QRS_NEXT_CUT()
PTP {E1 35457.209,E2 35457.209}
PTP {X 0,Y 759.903,A -85,B 0,C 180,E1 35457.209,E2 35457.209,E3 0,E4 0,E5 0,E6 0}
QRS_SPEED_INIT()
LIN {X 0,Y 759.903,Z 1305,A -85,B 0,C 180,E1 35457.209,E2 35457.209,E3 0,E4 0,E5 0,E6 0} C_VEL
LIN {X 0,Y 759.903,Z 603.404,A -85,B 0,C 180,E1 35457.209,E2 35457.209} C_VEL
LIN {X 0,Y 759.903,Z 595.326,A -85,B 0,C 180,E1 35457.209,E2 35457.209} C_VEL
LIN {X 0,Y 759.893,Z 593.326,A -85,B 0,C 180,E1 35457.058,E2 35457.058} C_VEL
LIN {X 0,Y 759.912,Z 593.326,A -85,B 0,C 180,E1 35454.261,E2 35454.261} C_VEL
LIN {X 0,Y 759.899,Z 593.323,A -85,B 0,C 180,E1 35451.373,E2 35451.373} C_VEL
LIN {X 0,Y 759.889,Z 593.322,A -85,B 0,C 180,E1 35448.539,E2 35448.539} C_VEL
LIN {X 0,Y 759.901,Z 593.322,A -85,B 0,C 180,E1 35445.756,E2 35445.756} C_VEL
LIN {X 0,Y 759.919,Z 593.324,A -85,B 0,C 180,E1 35442.858,E2 35442.858} C_VEL
LIN {X 0,Y 759.909,Z 593.326,A -85,B 0,C 180,E1 35439.96,E2 35439.96} C_VEL
LIN {X 0,Y 759.889,Z 593.323,A -85,B 0,C 180,E1 35437.159,E2 35437.159} C_VEL
LIN {X 0,Y 759.903,Z 593.32,A -85,B 0,C 180,E1 35434.33,E2 35434.33} C_VEL
LIN {X 0,Y 759.916,Z 593.32,A -85,B 0,C 180,E1 35431.354,E2 35431.354} C_VEL
LIN {X 0,Y 759.914,Z 593.321,A -85,B 0,C 180,E1 35428.331,E2 35428.331} C_VEL
LIN {X 0,Y 759.905,Z 593.327,A -85,B 0,C 180,E1 35425.451,E2 35425.451} C_VEL
LIN {X 0,Y 759.89,Z 593.326,A -85,B 0,C 180,E1 35422.656,E2 35422.656} C_VEL
LIN {X 0,Y 759.912,Z 593.32,A -85,B 0,C 180,E1 35419.853,E2 35419.853} C_VEL
LIN {X 0,Y 759.91,Z 593.319,A -85,B 0,C 180,E1 35416.826,E2 35416.826} C_VEL
LIN {X 0,Y 759.911,Z 593.32,A -85,B 0,C 180,E1 35413.795,E2 35413.795} C_VEL
LIN {X 0,Y 759.892,Z 593.325,A -85,B 0,C 180,E1 35410.939,E2 35410.939} C_VEL
LIN {X 0,Y 759.898,Z 593.327,A -85,B 0,C 180,E1 35408.2,E2 35408.2} C_VEL
LIN {X 0,Y 759.916,Z 593.321,A -85,B 0,C 180,E1 35405.282,E2 35405.282} C_VEL
LIN {X 0,Y 759.911,Z 593.32,A -85,B 0,C 180,E1 35402.289,E2 35402.289} C_VEL
LIN {X 0,Y 759.904,Z 593.321,A -85,B 0,C 180,E1 35399.305,E2 35399.305} C_VEL
LIN {X 0,Y 759.909,Z 593.575,A -85,B 0,C 180,E1 35398.059,E2 35398.059} C_VEL
LIN {X 0,Y 759.899,Z 638.776,A -85,B 0,C 180,E1 35395.191,E2 35395.191} C_VEL
LIN {X 0,Y 759.89,Z 682.695,A -85,B 0,C 180,E1 35392.472,E2 35392.472} C_VEL
LIN {X 0,Y 759.915,Z 727.991,A -85,B 0,C 180,E1 35389.723,E2 35389.723} C_VEL
LIN {X 0,Y 759.912,Z 778.002,A -85,B 0,C 180,E1 35386.746,E2 35386.746} C_VEL
LIN {X 0,Y 759.9,Z 826.73,A -85,B 0,C 180,E1 35383.893,E2 35383.893} C_VEL
LIN {X 0,Y 759.916,Z 830.801,A -85,B 0,C 180,E1 35383.665,E2 35383.665} C_VEL
LIN {X 0,Y 759.906,Z 999.951,A -85,B 0,C 180,E1 35382.036,E2 35382.036} C_VEL
LIN {X 0,Y 759.914,Z 1017.524,A -85,B 0,C 180,E1 35381.728,E2 35381.728} C_VEL
LIN {X 0,Y 759.905,Z 1033.905,A -85,B 0,C 180,E1 35381.305,E2 35381.305} C_VEL
LIN {X 0,Y 759.911,Z 1050.473,A -85,B 0,C 180,E1 35380.729,E2 35380.729} C_VEL
LIN {X 0,Y 759.918,Z 1065.925,A -85,B 0,C 180,E1 35380.039,E2 35380.039} C_VEL
LIN {X 0,Y 759.918,Z 1080.253,A -85,B 0,C 180,E1 35379.236,E2 35379.236} C_VEL
LIN {X 0,Y 759.918,Z 1093.584,A -85,B 0,C 180,E1 35378.319,E2 35378.319} C_VEL
LIN {X 0,Y 759.918,Z 1105.366,A -85,B 0,C 180,E1 35377.332,E2 35377.332} C_VEL
LIN {X 0,Y 759.919,Z 1115.725,A -85,B 0,C 180,E1 35376.269,E2 35376.269} C_VEL
LIN {X 0,Y 759.915,Z 1124.926,A -85,B 0,C 180,E1 35375.088,E2 35375.088} C_VEL
LIN {X 0,Y 759.916,Z 1132.481,A -85,B 0,C 180,E1 35373.847,E2 35373.847} C_VEL
LIN {X 0,Y 759.914,Z 1138.296,A -85,B 0,C 180,E1 35372.563,E2 35372.563} C_VEL
LIN {X 0,Y 759.913,Z 1142.253,A -85,B 0,C 180,E1 35371.281,E2 35371.281} C_VEL
LIN {X 0,Y 759.916,Z 1144.493,A -85,B 0,C 180,E1 35369.924,E2 35369.924} C_VEL
LIN {X 0,Y 759.915,Z 1144.892,A -85,B 0,C 180,E1 35368.566,E2 35368.566} C_VEL
LIN {X 0,Y 759.912,Z 1143.454,A -85,B 0,C 180,E1 35367.208,E2 35367.208} C_VEL
LIN {X 0,Y 759.918,Z 1140.29,A -85,B 0,C 180,E1 35365.925,E2 35365.925} C_VEL
LIN {X 0,Y 759.914,Z 1135.319,A -85,B 0,C 180,E1 35364.639,E2 35364.639} C_VEL
LIN {X 0,Y 759.914,Z 1128.391,A -85,B 0,C 180,E1 35363.35,E2 35363.35} C_VEL
LIN {X 0,Y 759.916,Z 1119.844,A -85,B 0,C 180,E1 35362.134,E2 35362.134} C_VEL
LIN {X 0,Y 759.917,Z 1109.619,A -85,B 0,C 180,E1 35360.991,E2 35360.991} C_VEL
LIN {X 0,Y 759.917,Z 1097.777,A -85,B 0,C 180,E1 35359.92,E2 35359.92} C_VEL
LIN {X 0,Y 759.917,Z 1085.153,A -85,B 0,C 180,E1 35358.987,E2 35358.987} C_VEL
LIN {X 0,Y 759.918,Z 1071.315,A -85,B 0,C 180,E1 35358.154,E2 35358.154} C_VEL
LIN {X 0,Y 759.913,Z 1056.24,A -85,B 0,C 180,E1 35357.421,E2 35357.421} C_VEL
LIN {X 0,Y 759.91,Z 1039.961,A -85,B 0,C 180,E1 35356.797,E2 35356.797} C_VEL
LIN {X 0,Y 759.908,Z 1023.505,A -85,B 0,C 180,E1 35356.318,E2 35356.318} C_VEL
LIN {X 0,Y 759.909,Z 1006.36,A -85,B 0,C 180,E1 35355.969,E2 35355.969} C_VEL
LIN {X 0,Y 759.906,Z 987.058,A -85,B 0,C 180,E1 35355.735,E2 35355.735} C_VEL
LIN {X 0,Y 759.911,Z 830.448,A -85,B 0,C 180,E1 35354.233,E2 35354.233} C_VEL
LIN {X 0,Y 759.914,Z 779.85,A -85,B 0,C 180,E1 35351.273,E2 35351.273} C_VEL
LIN {X 0,Y 759.905,Z 729.874,A -85,B 0,C 180,E1 35348.299,E2 35348.299} C_VEL
LIN {X 0,Y 759.889,Z 684.484,A -85,B 0,C 180,E1 35345.548,E2 35345.548} C_VEL
LIN {X 0,Y 759.904,Z 640.226,A -85,B 0,C 180,E1 35342.81,E2 35342.81} C_VEL
LIN {X 0,Y 759.907,Z 594.516,A -85,B 0,C 180,E1 35339.912,E2 35339.912} C_VEL
LIN {X 0,Y 759.91,Z 593.318,A -85,B 0,C 180,E1 35339.824,E2 35339.824} C_VEL
LIN {X 0,Y 759.915,Z 593.322,A -85,B 0,C 180,E1 35336.809,E2 35336.809} C_VEL
LIN {X 0,Y 759.891,Z 593.317,A -85,B 0,C 180,E1 35333.972,E2 35333.972} C_VEL
LIN {X 0,Y 759.918,Z 593.327,A -85,B 0,C 180,E1 35331.124,E2 35331.124} C_VEL
LIN {X 0,Y 759.906,Z 593.315,A -85,B 0,C 180,E1 35328.251,E2 35328.251} C_VEL
LIN {X 0,Y 759.913,Z 593.328,A -85,B 0,C 180,E1 35325.255,E2 35325.255} C_VEL
LIN {X 0,Y 759.906,Z 593.315,A -85,B 0,C 180,E1 35322.251,E2 35322.251} C_VEL
LIN {X 0,Y 759.91,Z 593.328,A -85,B 0,C 180,E1 35319.313,E2 35319.313} C_VEL
LIN {X 0,Y 759.889,Z 593.318,A -85,B 0,C 180,E1 35316.488,E2 35316.488} C_VEL
LIN {X 0,Y 759.914,Z 593.324,A -85,B 0,C 180,E1 35313.602,E2 35313.602} C_VEL
LIN {X 0,Y 759.911,Z 593.315,A -85,B 0,C 180,E1 35310.612,E2 35310.612} C_VEL
LIN {X 0,Y 759.918,Z 593.327,A -85,B 0,C 180,E1 35307.591,E2 35307.591} C_VEL
LIN {X 0,Y 759.91,Z 593.353,A -85,B 0,C 180,E1 35306.575,E2 35306.575} C_VEL
LIN {X 0,Y 759.889,Z 601.331,A -85,B 0,C 180,E1 35305.967,E2 35305.967} C_VEL
LIN {X 0,Y 759.915,Z 858.573,A -85,B 0,C 180,E1 35303.276,E2 35303.276} C_VEL
LIN {X 0,Y 759.913,Z 946.529,A -85,B 0,C 180,E1 35302.35,E2 35302.35} C_VEL
LIN {X 0,Y 759.909,Z 970.175,A -85,B 0,C 180,E1 35301.964,E2 35301.964} C_VEL
LIN {X 0,Y 759.908,Z 991.488,A -85,B 0,C 180,E1 35301.489,E2 35301.489} C_VEL
LIN {X 0,Y 759.898,Z 1013.758,A -85,B 0,C 180,E1 35300.851,E2 35300.851} C_VEL
LIN {X 0,Y 759.918,Z 1033.44,A -85,B 0,C 180,E1 35300.166,E2 35300.166} C_VEL
LIN {X 0,Y 759.919,Z 1054.673,A -85,B 0,C 180,E1 35299.285,E2 35299.285} C_VEL
LIN {X 0,Y 759.914,Z 1074.389,A -85,B 0,C 180,E1 35298.329,E2 35298.329} C_VEL
LIN {X 0,Y 759.917,Z 1093.916,A -85,B 0,C 180,E1 35297.221,E2 35297.221} C_VEL
LIN {X 0,Y 759.911,Z 1112.133,A -85,B 0,C 180,E1 35296.041,E2 35296.041} C_VEL
LIN {X 0,Y 759.913,Z 1129.871,A -85,B 0,C 180,E1 35294.711,E2 35294.711} C_VEL
LIN {X 0,Y 759.909,Z 1146.093,A -85,B 0,C 180,E1 35293.313,E2 35293.313} C_VEL
LIN {X 0,Y 759.909,Z 1161,A -85,B 0,C 180,E1 35291.845,E2 35291.845} C_VEL
LIN {X 0,Y 759.899,Z 1173.75,A -85,B 0,C 180,E1 35290.385,E2 35290.385} C_VEL
LIN {X 0,Y 759.909,Z 1186.404,A -85,B 0,C 180,E1 35288.703,E2 35288.703} C_VEL
LIN {X 0,Y 759.911,Z 1196.1,A -85,B 0,C 180,E1 35287.181,E2 35287.181} C_VEL
LIN {X 0,Y 759.896,Z 1205.307,A -85,B 0,C 180,E1 35285.436,E2 35285.436} C_VEL
LIN {X 0,Y 759.903,Z 1211.799,A -85,B 0,C 180,E1 35283.923,E2 35283.923} C_VEL
LIN {X 0,Y 759.915,Z 1217.779,A -85,B 0,C 180,E1 35282.111,E2 35282.111} C_VEL
LIN {X 0,Y 759.917,Z 1221.69,A -85,B 0,C 180,E1 35280.452,E2 35280.452} C_VEL
LIN {X 0,Y 759.91,Z 1224.098,A -85,B 0,C 180,E1 35278.718,E2 35278.718} C_VEL
LIN {X 0,Y 759.909,Z 1224.976,A -85,B 0,C 180,E1 35277.058,E2 35277.058} C_VEL
LIN {X 0,Y 759.91,Z 1224.211,A -85,B 0,C 180,E1 35275.321,E2 35275.321} C_VEL
LIN {X 0,Y 759.894,Z 1221.944,A -85,B 0,C 180,E1 35273.578,E2 35273.578} C_VEL
LIN {X 0,Y 759.917,Z 1218.072,A -85,B 0,C 180,E1 35271.906,E2 35271.906} C_VEL
LIN {X 0,Y 759.914,Z 1212.453,A -85,B 0,C 180,E1 35270.151,E2 35270.151} C_VEL
LIN {X 0,Y 759.906,Z 1205.614,A -85,B 0,C 180,E1 35268.54,E2 35268.54} C_VEL
LIN {X 0,Y 759.914,Z 1196.782,A -85,B 0,C 180,E1 35266.842,E2 35266.842} C_VEL
LIN {X 0,Y 759.897,Z 1186.955,A -85,B 0,C 180,E1 35265.288,E2 35265.288} C_VEL
LIN {X 0,Y 759.907,Z 1174.745,A -85,B 0,C 180,E1 35263.645,E2 35263.645} C_VEL
LIN {X 0,Y 759.914,Z 1162.457,A -85,B 0,C 180,E1 35262.226,E2 35262.226} C_VEL
LIN {X 0,Y 759.916,Z 1147.367,A -85,B 0,C 180,E1 35260.715,E2 35260.715} C_VEL
LIN {X 0,Y 759.915,Z 1131.348,A -85,B 0,C 180,E1 35259.314,E2 35259.314} C_VEL
LIN {X 0,Y 759.917,Z 1113.604,A -85,B 0,C 180,E1 35257.976,E2 35257.976} C_VEL
LIN {X 0,Y 759.917,Z 1094.916,A -85,B 0,C 180,E1 35256.75,E2 35256.75} C_VEL
LIN {X 0,Y 759.919,Z 1076.273,A -85,B 0,C 180,E1 35255.679,E2 35255.679} C_VEL
LIN {X 0,Y 759.916,Z 1055.929,A -85,B 0,C 180,E1 35254.682,E2 35254.682} C_VEL
LIN {X 0,Y 759.918,Z 1034.648,A -85,B 0,C 180,E1 35253.788,E2 35253.788} C_VEL
LIN {X 0,Y 759.902,Z 1014.583,A -85,B 0,C 180,E1 35253.087,E2 35253.087} C_VEL
LIN {X 0,Y 759.918,Z 993.181,A -85,B 0,C 180,E1 35252.462,E2 35252.462} C_VEL
LIN {X 0,Y 759.906,Z 971.975,A -85,B 0,C 180,E1 35251.982,E2 35251.982} C_VEL
LIN {X 0,Y 759.915,Z 949.573,A -85,B 0,C 180,E1 35251.598,E2 35251.598} C_VEL
LIN {X 0,Y 759.914,Z 903.373,A -85,B 0,C 180,E1 35251.095,E2 35251.095} C_VEL
LIN {X 0,Y 759.913,Z 631.659,A -85,B 0,C 180,E1 35248.265,E2 35248.265} C_VEL
LIN {X 0,Y 759.893,Z 600.869,A -85,B 0,C 180,E1 35247.93,E2 35247.93} C_VEL
LIN {X 0,Y 759.911,Z 593.322,A -85,B 0,C 180,E1 35247.307,E2 35247.307} C_VEL
LIN {X 0,Y 759.897,Z 593.322,A -85,B 0,C 180,E1 35244.344,E2 35244.344} C_VEL
LIN {X 0,Y 759.891,Z 593.324,A -85,B 0,C 180,E1 35241.529,E2 35241.529} C_VEL
LIN {X 0,Y 759.902,Z 593.328,A -85,B 0,C 180,E1 35238.706,E2 35238.706} C_VEL
LIN {X 0,Y 759.913,Z 593.325,A -85,B 0,C 180,E1 35236.888,E2 35236.888} C_VEL
LIN {X 0,Y 759.918,Z 654.539,A -85,B 0,C 180,E1 35234.851,E2 35234.851} C_VEL
LIN {X 0,Y 759.92,Z 699.236,A -85,B 0,C 180,E1 35233.202,E2 35233.202} C_VEL
LIN {X 0,Y 759.92,Z 738.808,A -85,B 0,C 180,E1 35231.589,E2 35231.589} C_VEL
LIN {X 0,Y 759.917,Z 752.824,A -85,B 0,C 180,E1 35230.89,E2 35230.89} C_VEL
LIN {X 0,Y 759.908,Z 764.753,A -85,B 0,C 180,E1 35230.139,E2 35230.139} C_VEL
LIN {X 0,Y 759.908,Z 773.509,A -85,B 0,C 180,E1 35229.432,E2 35229.432} C_VEL
LIN {X 0,Y 759.893,Z 779.468,A -85,B 0,C 180,E1 35228.781,E2 35228.781} C_VEL
LIN {X 0,Y 759.895,Z 782.672,A -85,B 0,C 180,E1 35228.203,E2 35228.203} C_VEL
LIN {X 0,Y 759.891,Z 783.283,A -85,B 0,C 180,E1 35227.82,E2 35227.82} C_VEL
LIN {X 0,Y 759.909,Z 782.173,A -85,B 0,C 180,E1 35227.493,E2 35227.493} C_VEL
LIN {X 0,Y 759.899,Z 779.495,A -85,B 0,C 180,E1 35227.243,E2 35227.243} C_VEL
LIN {X 0,Y 759.891,Z 775.795,A -85,B 0,C 180,E1 35227.089,E2 35227.089} C_VEL
LIN {X 0,Y 759.889,Z 769.468,A -85,B 0,C 180,E1 35226.992,E2 35226.992} C_VEL
LIN {X 0,Y 759.889,Z 593.325,A -85,B 0,C 180,E1 35226.966,E2 35226.966} C_VEL
LIN {X 0,Y 759.9,Z 593.351,A -85,B 0,C 180,E1 35224.136,E2 35224.136} C_VEL
LIN {X 0,Y 759.915,Z 633.667,A -85,B 0,C 180,E1 35221.404,E2 35221.404} C_VEL
LIN {X 0,Y 759.908,Z 669.855,A -85,B 0,C 180,E1 35219.026,E2 35219.026} C_VEL
LIN {X 0,Y 759.91,Z 945.711,A -85,B 0,C 180,E1 35216.145,E2 35216.145} C_VEL
LIN {X 0,Y 759.903,Z 1017.761,A -85,B 0,C 180,E1 35215.381,E2 35215.381} C_VEL
LIN {X 0,Y 759.916,Z 1040.309,A -85,B 0,C 180,E1 35215.006,E2 35215.006} C_VEL
LIN {X 0,Y 759.901,Z 1060.837,A -85,B 0,C 180,E1 35214.55,E2 35214.55} C_VEL
LIN {X 0,Y 759.918,Z 1083.358,A -85,B 0,C 180,E1 35213.908,E2 35213.908} C_VEL
LIN {X 0,Y 759.919,Z 1103.501,A -85,B 0,C 180,E1 35213.209,E2 35213.209} C_VEL
LIN {X 0,Y 759.917,Z 1124.653,A -85,B 0,C 180,E1 35212.331,E2 35212.331} C_VEL
LIN {X 0,Y 759.913,Z 1144.352,A -85,B 0,C 180,E1 35211.376,E2 35211.376} C_VEL
LIN {X 0,Y 759.913,Z 1163.511,A -85,B 0,C 180,E1 35210.291,E2 35210.291} C_VEL
LIN {X 0,Y 759.912,Z 1182.127,A -85,B 0,C 180,E1 35209.086,E2 35209.086} C_VEL
LIN {X 0,Y 759.913,Z 1199.122,A -85,B 0,C 180,E1 35207.814,E2 35207.814} C_VEL
LIN {X 0,Y 759.908,Z 1215.45,A -85,B 0,C 180,E1 35206.418,E2 35206.418} C_VEL
LIN {X 0,Y 759.902,Z 1230.487,A -85,B 0,C 180,E1 35204.946,E2 35204.946} C_VEL
LIN {X 0,Y 759.916,Z 1243.43,A -85,B 0,C 180,E1 35203.468,E2 35203.468} C_VEL
LIN {X 0,Y 759.912,Z 1255.749,A -85,B 0,C 180,E1 35201.846,E2 35201.846} C_VEL
LIN {X 0,Y 759.908,Z 1265.598,A -85,B 0,C 180,E1 35200.309,E2 35200.309} C_VEL
LIN {X 0,Y 759.9,Z 1274.979,A -85,B 0,C 180,E1 35198.552,E2 35198.552} C_VEL
LIN {X 0,Y 759.905,Z 1281.552,A -85,B 0,C 180,E1 35197.03,E2 35197.03} C_VEL
LIN {X 0,Y 759.914,Z 1287.635,A -85,B 0,C 180,E1 35195.21,E2 35195.21} C_VEL
LIN {X 0,Y 759.892,Z 1291.43,A -85,B 0,C 180,E1 35193.622,E2 35193.622} C_VEL
LIN {X 0,Y 759.9,Z 1294.056,A -85,B 0,C 180,E1 35191.811,E2 35191.811} C_VEL
LIN {X 0,Y 759.905,Z 1294.962,A -85,B 0,C 180,E1 35190.152,E2 35190.152} C_VEL
LIN {X 0,Y 759.891,Z 1294.258,A -85,B 0,C 180,E1 35188.418,E2 35188.418} C_VEL
LIN {X 0,Y 759.902,Z 1292.055,A -85,B 0,C 180,E1 35186.682,E2 35186.682} C_VEL
LIN {X 0,Y 759.912,Z 1288.051,A -85,B 0,C 180,E1 35184.943,E2 35184.943} C_VEL
LIN {X 0,Y 759.893,Z 1282.47,A -85,B 0,C 180,E1 35183.2,E2 35183.2} C_VEL
LIN {X 0,Y 759.909,Z 1275.698,A -85,B 0,C 180,E1 35181.603,E2 35181.603} C_VEL
LIN {X 0,Y 759.914,Z 1266.996,A -85,B 0,C 180,E1 35179.923,E2 35179.923} C_VEL
LIN {X 0,Y 759.912,Z 1257.319,A -85,B 0,C 180,E1 35178.387,E2 35178.387} C_VEL
LIN {X 0,Y 759.909,Z 1245.37,A -85,B 0,C 180,E1 35176.766,E2 35176.766} C_VEL
LIN {X 0,Y 759.912,Z 1232.63,A -85,B 0,C 180,E1 35175.29,E2 35175.29} C_VEL
LIN {X 0,Y 759.917,Z 1217.845,A -85,B 0,C 180,E1 35173.804,E2 35173.804} C_VEL
LIN {X 0,Y 759.918,Z 1201.68,A -85,B 0,C 180,E1 35172.386,E2 35172.386} C_VEL
LIN {X 0,Y 759.914,Z 1184.643,A -85,B 0,C 180,E1 35171.096,E2 35171.096} C_VEL
LIN {X 0,Y 759.916,Z 1165.59,A -85,B 0,C 180,E1 35169.836,E2 35169.836} C_VEL
LIN {X 0,Y 759.916,Z 1146.708,A -85,B 0,C 180,E1 35168.748,E2 35168.748} C_VEL
LIN {X 0,Y 759.915,Z 1126.937,A -85,B 0,C 180,E1 35167.774,E2 35167.774} C_VEL
LIN {X 0,Y 759.919,Z 1106.136,A -85,B 0,C 180,E1 35166.888,E2 35166.888} C_VEL
LIN {X 0,Y 759.915,Z 1085.288,A -85,B 0,C 180,E1 35166.154,E2 35166.154} C_VEL
LIN {X 0,Y 759.904,Z 1063.504,A -85,B 0,C 180,E1 35165.515,E2 35165.515} C_VEL
LIN {X 0,Y 759.919,Z 1042.443,A -85,B 0,C 180,E1 35165.037,E2 35165.037} C_VEL
LIN {X 0,Y 759.905,Z 1020.366,A -85,B 0,C 180,E1 35164.653,E2 35164.653} C_VEL
LIN {X 0,Y 759.903,Z 979.523,A -85,B 0,C 180,E1 35164.203,E2 35164.203} C_VEL
LIN {X 0,Y 759.904,Z 721.424,A -85,B 0,C 180,E1 35161.518,E2 35161.518} C_VEL
LIN {X 0,Y 759.91,Z 669.44,A -85,B 0,C 180,E1 35160.954,E2 35160.954} C_VEL
LIN {X 0,Y 759.9,Z 627.085,A -85,B 0,C 180,E1 35158.155,E2 35158.155} C_VEL
LIN {X 0,Y 759.901,Z 593.323,A -85,B 0,C 180,E1 35155.858,E2 35155.858} C_VEL
LIN {X 0,Y 759.889,Z 593.325,A -85,B 0,C 180,E1 35153.016,E2 35153.016} C_VEL
LIN {X 0,Y 759.889,Z 770.611,A -85,B 0,C 180,E1 35153,E2 35153} C_VEL
LIN {X 0,Y 759.892,Z 776.724,A -85,B 0,C 180,E1 35152.882,E2 35152.882} C_VEL
LIN {X 0,Y 759.903,Z 780.253,A -85,B 0,C 180,E1 35152.706,E2 35152.706} C_VEL
LIN {X 0,Y 759.908,Z 782.413,A -85,B 0,C 180,E1 35152.469,E2 35152.469} C_VEL
LIN {X 0,Y 759.89,Z 783.298,A -85,B 0,C 180,E1 35152.139,E2 35152.139} C_VEL
LIN {X 0,Y 759.903,Z 782.303,A -85,B 0,C 180,E1 35151.704,E2 35151.704} C_VEL
LIN {X 0,Y 759.89,Z 778.75,A -85,B 0,C 180,E1 35151.125,E2 35151.125} C_VEL
LIN {X 0,Y 759.916,Z 772.144,A -85,B 0,C 180,E1 35150.445,E2 35150.445} C_VEL
LIN {X 0,Y 759.917,Z 762.445,A -85,B 0,C 180,E1 35149.701,E2 35149.701} C_VEL
LIN {X 0,Y 759.913,Z 722.491,A -85,B 0,C 180,E1 35146.932,E2 35146.932} C_VEL
LIN {X 0,Y 759.919,Z 684.652,A -85,B 0,C 180,E1 35144.216,E2 35144.216} C_VEL
LIN {X 0,Y 759.912,Z 648.559,A -85,B 0,C 180,E1 35141.526,E2 35141.526} C_VEL
LIN {X 0,Y 759.916,Z 613.129,A -85,B 0,C 180,E1 35138.779,E2 35138.779} C_VEL
LIN {X 0,Y 759.9,Z 593.329,A -85,B 0,C 180,E1 35137.177,E2 35137.177} C_VEL
LIN {X 0,Y 759.892,Z 593.323,A -85,B 0,C 180,E1 35134.367,E2 35134.367} C_VEL
LIN {X 0,Y 759.904,Z 593.321,A -85,B 0,C 180,E1 35131.58,E2 35131.58} C_VEL
LIN {X 0,Y 759.918,Z 593.32,A -85,B 0,C 180,E1 35128.617,E2 35128.617} C_VEL
LIN {X 0,Y 759.904,Z 593.324,A -85,B 0,C 180,E1 35125.652,E2 35125.652} C_VEL
LIN {X 0,Y 759.91,Z 593.328,A -85,B 0,C 180,E1 35122.758,E2 35122.758} C_VEL
LIN {X 0,Y 759.905,Z 593.323,A -85,B 0,C 180,E1 35119.925,E2 35119.925} C_VEL
LIN {X 0,Y 759.908,Z 593.32,A -85,B 0,C 180,E1 35117.063,E2 35117.063} C_VEL
LIN {X 0,Y 759.915,Z 593.319,A -85,B 0,C 180,E1 35114.089,E2 35114.089} C_VEL
LIN {X 0,Y 759.905,Z 593.321,A -85,B 0,C 180,E1 35111.076,E2 35111.076} C_VEL
LIN {X 0,Y 759.908,Z 593.323,A -85,B 0,C 180,E1 35108.17,E2 35108.17} C_VEL
LIN {X 0,Y 759.917,Z 593.327,A -85,B 0,C 180,E1 35105.285,E2 35105.285} C_VEL
LIN {X 0,Y 759.901,Z 593.324,A -85,B 0,C 180,E1 35102.413,E2 35102.413} C_VEL
LIN {X 0,Y 759.916,Z 593.32,A -85,B 0,C 180,E1 35099.472,E2 35099.472} C_VEL
LIN {X 0,Y 759.893,Z 593.326,A -85,B 0,C 180,E1 35097.058,E2 35097.058} C_VEL
LIN {X 0,Y 758.883,Z 593.45,A -85,B 0,C 180,E1 35096.477,E2 35096.477} C_VEL
LIN {X 0,Y 752.477,Z 594.247,A -85,B 0,C 180,E1 35094.851,E2 35094.851} C_VEL
LIN {X 0,Y 751.966,Z 594.313,A -85,B 0,C 180,E1 35094.428,E2 35094.428} C_VEL
LIN {X 0,Y 751.951,Z 594.311,A -85,B 0,C 180,E1 35091.589,E2 35091.589} C_VEL
LIN {X 0,Y 751.958,Z 594.311,A -85,B 0,C 180,E1 35088.806,E2 35088.806} C_VEL
LIN {X 0,Y 751.974,Z 594.312,A -85,B 0,C 180,E1 35085.917,E2 35085.917} C_VEL
LIN {X 0,Y 751.975,Z 594.316,A -85,B 0,C 180,E1 35082.99,E2 35082.99} C_VEL
LIN {X 0,Y 751.965,Z 594.314,A -85,B 0,C 180,E1 35080.063,E2 35080.063} C_VEL
LIN {X 0,Y 751.952,Z 594.312,A -85,B 0,C 180,E1 35077.235,E2 35077.235} C_VEL
LIN {X 0,Y 751.966,Z 594.309,A -85,B 0,C 180,E1 35074.357,E2 35074.357} C_VEL
LIN {X 0,Y 751.977,Z 594.309,A -85,B 0,C 180,E1 35071.349,E2 35071.349} C_VEL
LIN {X 0,Y 751.976,Z 594.31,A -85,B 0,C 180,E1 35068.316,E2 35068.316} C_VEL
LIN {X 0,Y 751.963,Z 594.315,A -85,B 0,C 180,E1 35065.392,E2 35065.392} C_VEL
LIN {X 0,Y 751.954,Z 594.316,A -85,B 0,C 180,E1 35062.578,E2 35062.578} C_VEL
LIN {X 0,Y 751.967,Z 594.31,A -85,B 0,C 180,E1 35059.741,E2 35059.741} C_VEL
LIN {X 0,Y 751.972,Z 594.307,A -85,B 0,C 180,E1 35056.773,E2 35056.773} C_VEL
LIN {X 0,Y 751.975,Z 594.308,A -85,B 0,C 180,E1 35053.742,E2 35053.742} C_VEL
LIN {X 0,Y 751.966,Z 594.31,A -85,B 0,C 180,E1 35050.718,E2 35050.718} C_VEL
LIN {X 0,Y 751.971,Z 594.312,A -85,B 0,C 180,E1 35047.804,E2 35047.804} C_VEL
LIN {X 0,Y 751.975,Z 594.316,A -85,B 0,C 180,E1 35044.872,E2 35044.872} C_VEL
LIN {X 0,Y 751.956,Z 594.315,A -85,B 0,C 180,E1 35041.966,E2 35041.966} C_VEL
LIN {X 0,Y 751.976,Z 594.311,A -85,B 0,C 180,E1 35039.033,E2 35039.033} C_VEL
LIN {X 0,Y 751.978,Z 594.46,A -85,B 0,C 180,E1 35038.338,E2 35038.338} C_VEL
LIN {X 0,Y 752.539,Z 597.101,A -85,B 0,C 180,E1 35038.142,E2 35038.142} C_VEL
LIN {X 0,Y 752.435,Z 643.633,A -85,B 0,C 180,E1 35035.164,E2 35035.164} C_VEL
LIN {X 0,Y 752.308,Z 690.886,A -85,B 0,C 180,E1 35032.216,E2 35032.216} C_VEL
LIN {X 0,Y 752.23,Z 737.522,A -85,B 0,C 180,E1 35029.367,E2 35029.367} C_VEL
LIN {X 0,Y 752.134,Z 784.873,A -85,B 0,C 180,E1 35026.527,E2 35026.527} C_VEL
LIN {X 0,Y 752.127,Z 831.04,A -85,B 0,C 180,E1 35023.819,E2 35023.819} C_VEL
LIN {X 0,Y 752.109,Z 1000.901,A -85,B 0,C 180,E1 35022.161,E2 35022.161} C_VEL
LIN {X 0,Y 752.098,Z 1018.47,A -85,B 0,C 180,E1 35021.842,E2 35021.842} C_VEL
LIN {X 0,Y 752.065,Z 1035.556,A -85,B 0,C 180,E1 35021.386,E2 35021.386} C_VEL
LIN {X 0,Y 752.045,Z 1051.749,A -85,B 0,C 180,E1 35020.804,E2 35020.804} C_VEL
LIN {X 0,Y 752.022,Z 1066.89,A -85,B 0,C 180,E1 35020.107,E2 35020.107} C_VEL
LIN {X 0,Y 751.995,Z 1081.634,A -85,B 0,C 180,E1 35019.257,E2 35019.257} C_VEL
LIN {X 0,Y 751.972,Z 1095.224,A -85,B 0,C 180,E1 35018.294,E2 35018.294} C_VEL
LIN {X 0,Y 751.95,Z 1107.091,A -85,B 0,C 180,E1 35017.256,E2 35017.256} C_VEL
LIN {X 0,Y 751.936,Z 1117.73,A -85,B 0,C 180,E1 35016.106,E2 35016.106} C_VEL
LIN {X 0,Y 751.925,Z 1126.76,A -85,B 0,C 180,E1 35014.881,E2 35014.881} C_VEL
LIN {X 0,Y 751.917,Z 1133.743,A -85,B 0,C 180,E1 35013.659,E2 35013.659} C_VEL
LIN {X 0,Y 751.916,Z 1139.155,A -85,B 0,C 180,E1 35012.362,E2 35012.362} C_VEL
LIN {X 0,Y 751.915,Z 1142.75,A -85,B 0,C 180,E1 35011.066,E2 35011.066} C_VEL
LIN {X 0,Y 751.911,Z 1144.701,A -85,B 0,C 180,E1 35009.694,E2 35009.694} C_VEL
LIN {X 0,Y 751.914,Z 1144.844,A -85,B 0,C 180,E1 35008.399,E2 35008.399} C_VEL
LIN {X 0,Y 751.916,Z 1143.181,A -85,B 0,C 180,E1 35007.054,E2 35007.054} C_VEL
LIN {X 0,Y 751.916,Z 1139.749,A -85,B 0,C 180,E1 35005.728,E2 35005.728} C_VEL
LIN {X 0,Y 751.918,Z 1134.564,A -85,B 0,C 180,E1 35004.428,E2 35004.428} C_VEL
LIN {X 0,Y 751.922,Z 1127.865,A -85,B 0,C 180,E1 35003.202,E2 35003.202} C_VEL
LIN {X 0,Y 751.931,Z 1119.755,A -85,B 0,C 180,E1 35002.05,E2 35002.05} C_VEL
LIN {X 0,Y 751.946,Z 1109.508,A -85,B 0,C 180,E1 35000.894,E2 35000.894} C_VEL
LIN {X 0,Y 751.965,Z 1097.643,A -85,B 0,C 180,E1 34999.813,E2 34999.813} C_VEL
LIN {X 0,Y 751.991,Z 1084.604,A -85,B 0,C 180,E1 34998.844,E2 34998.844} C_VEL
LIN {X 0,Y 752.018,Z 1070.374,A -85,B 0,C 180,E1 34997.989,E2 34997.989} C_VEL
LIN {X 0,Y 752.036,Z 1055.087,A -85,B 0,C 180,E1 34997.248,E2 34997.248} C_VEL
LIN {X 0,Y 752.061,Z 1038.686,A -85,B 0,C 180,E1 34996.623,E2 34996.623} C_VEL
LIN {X 0,Y 752.094,Z 1021.504,A -85,B 0,C 180,E1 34996.136,E2 34996.136} C_VEL
LIN {X 0,Y 752.109,Z 1003.819,A -85,B 0,C 180,E1 34995.793,E2 34995.793} C_VEL
LIN {X 0,Y 752.121,Z 979.09,A -85,B 0,C 180,E1 34995.52,E2 34995.52} C_VEL
LIN {X 0,Y 752.08,Z 830.586,A -85,B 0,C 180,E1 34994.084,E2 34994.084} C_VEL
LIN {X 0,Y 752.16,Z 780.324,A -85,B 0,C 180,E1 34991.112,E2 34991.112} C_VEL
LIN {X 0,Y 752.244,Z 729.672,A -85,B 0,C 180,E1 34988.067,E2 34988.067} C_VEL
LIN {X 0,Y 752.313,Z 684.373,A -85,B 0,C 180,E1 34985.291,E2 34985.291} C_VEL
LIN {X 0,Y 752.42,Z 640.382,A -85,B 0,C 180,E1 34982.539,E2 34982.539} C_VEL
LIN {X 0,Y 752.542,Z 596.496,A -85,B 0,C 180,E1 34979.729,E2 34979.729} C_VEL
LIN {X 0,Y 751.958,Z 594.314,A -85,B 0,C 180,E1 34979.56,E2 34979.56} C_VEL
LIN {X 0,Y 751.972,Z 594.308,A -85,B 0,C 180,E1 34976.621,E2 34976.621} C_VEL
LIN {X 0,Y 751.967,Z 594.306,A -85,B 0,C 180,E1 34973.72,E2 34973.72} C_VEL
LIN {X 0,Y 751.968,Z 594.309,A -85,B 0,C 180,E1 34970.825,E2 34970.825} C_VEL
LIN {X 0,Y 751.953,Z 594.307,A -85,B 0,C 180,E1 34968.015,E2 34968.015} C_VEL
LIN {X 0,Y 751.97,Z 594.315,A -85,B 0,C 180,E1 34965.132,E2 34965.132} C_VEL
LIN {X 0,Y 751.972,Z 594.304,A -85,B 0,C 180,E1 34962.183,E2 34962.183} C_VEL
LIN {X 0,Y 751.974,Z 594.313,A -85,B 0,C 180,E1 34959.169,E2 34959.169} C_VEL
LIN {X 0,Y 751.952,Z 594.307,A -85,B 0,C 180,E1 34956.28,E2 34956.28} C_VEL
LIN {X 0,Y 751.97,Z 594.317,A -85,B 0,C 180,E1 34953.401,E2 34953.401} C_VEL
LIN {X 0,Y 751.962,Z 594.306,A -85,B 0,C 180,E1 34950.497,E2 34950.497} C_VEL
LIN {X 0,Y 751.974,Z 594.317,A -85,B 0,C 180,E1 34947.513,E2 34947.513} C_VEL
LIN {X 0,Y 751.955,Z 594.314,A -85,B 0,C 180,E1 34946.843,E2 34946.843} C_VEL
LIN {X 0,Y 752.456,Z 597.312,A -85,B 0,C 180,E1 34946.58,E2 34946.58} C_VEL
LIN {X 0,Y 752.51,Z 601.377,A -85,B 0,C 180,E1 34946.278,E2 34946.278} C_VEL
LIN {X 0,Y 752.885,Z 605.076,A -85,B 0,C 180,E1 34946.223,E2 34946.223} C_VEL
LIN {X 0,Y 752.737,Z 862.55,A -85,B 0,C 180,E1 34943.505,E2 34943.505} C_VEL
LIN {X 0,Y 752.677,Z 946.964,A -85,B 0,C 180,E1 34942.607,E2 34942.607} C_VEL
LIN {X 0,Y 752.626,Z 970.841,A -85,B 0,C 180,E1 34942.21,E2 34942.21} C_VEL
LIN {X 0,Y 752.581,Z 992.621,A -85,B 0,C 180,E1 34941.717,E2 34941.717} C_VEL
LIN {X 0,Y 752.495,Z 1014.836,A -85,B 0,C 180,E1 34941.065,E2 34941.065} C_VEL
LIN {X 0,Y 752.456,Z 1035.477,A -85,B 0,C 180,E1 34940.334,E2 34940.334} C_VEL
LIN {X 0,Y 752.375,Z 1056.309,A -85,B 0,C 180,E1 34939.446,E2 34939.446} C_VEL
LIN {X 0,Y 752.294,Z 1076.555,A -85,B 0,C 180,E1 34938.441,E2 34938.441} C_VEL
LIN {X 0,Y 752.231,Z 1095.783,A -85,B 0,C 180,E1 34937.323,E2 34937.323} C_VEL
LIN {X 0,Y 752.152,Z 1115.146,A -85,B 0,C 180,E1 34936.025,E2 34936.025} C_VEL
LIN {X 0,Y 752.097,Z 1132.251,A -85,B 0,C 180,E1 34934.71,E2 34934.71} C_VEL
LIN {X 0,Y 752.043,Z 1147.294,A -85,B 0,C 180,E1 34933.376,E2 34933.376} C_VEL
LIN {X 0,Y 751.995,Z 1162.703,A -85,B 0,C 180,E1 34931.816,E2 34931.816} C_VEL
LIN {X 0,Y 751.961,Z 1175.296,A -85,B 0,C 180,E1 34930.341,E2 34930.341} C_VEL
LIN {X 0,Y 751.944,Z 1187.14,A -85,B 0,C 180,E1 34928.719,E2 34928.719} C_VEL
LIN {X 0,Y 751.936,Z 1196.755,A -85,B 0,C 180,E1 34927.181,E2 34927.181} C_VEL
LIN {X 0,Y 751.908,Z 1205.462,A -85,B 0,C 180,E1 34925.494,E2 34925.494} C_VEL
LIN {X 0,Y 751.91,Z 1212.534,A -85,B 0,C 180,E1 34923.812,E2 34923.812} C_VEL
LIN {X 0,Y 751.916,Z 1217.865,A -85,B 0,C 180,E1 34922.134,E2 34922.134} C_VEL
LIN {X 0,Y 751.917,Z 1221.759,A -85,B 0,C 180,E1 34920.457,E2 34920.457} C_VEL
LIN {X 0,Y 751.911,Z 1224.129,A -85,B 0,C 180,E1 34918.705,E2 34918.705} C_VEL
LIN {X 0,Y 751.912,Z 1225,A -85,B 0,C 180,E1 34916.951,E2 34916.951} C_VEL
LIN {X 0,Y 751.907,Z 1224.118,A -85,B 0,C 180,E1 34915.194,E2 34915.194} C_VEL
LIN {X 0,Y 751.902,Z 1221.653,A -85,B 0,C 180,E1 34913.401,E2 34913.401} C_VEL
LIN {X 0,Y 751.912,Z 1217.779,A -85,B 0,C 180,E1 34911.743,E2 34911.743} C_VEL
LIN {X 0,Y 751.923,Z 1211.713,A -85,B 0,C 180,E1 34909.89,E2 34909.89} C_VEL
LIN {X 0,Y 751.915,Z 1205.107,A -85,B 0,C 180,E1 34908.338,E2 34908.338} C_VEL
LIN {X 0,Y 751.926,Z 1195.65,A -85,B 0,C 180,E1 34906.543,E2 34906.543} C_VEL
LIN {X 0,Y 751.943,Z 1186.203,A -85,B 0,C 180,E1 34905.05,E2 34905.05} C_VEL
LIN {X 0,Y 751.971,Z 1173.818,A -85,B 0,C 180,E1 34903.388,E2 34903.388} C_VEL
LIN {X 0,Y 752.009,Z 1160.714,A -85,B 0,C 180,E1 34901.872,E2 34901.872} C_VEL
LIN {X 0,Y 752.043,Z 1146.125,A -85,B 0,C 180,E1 34900.424,E2 34900.424} C_VEL
LIN {X 0,Y 752.102,Z 1129.834,A -85,B 0,C 180,E1 34899.005,E2 34899.005} C_VEL
LIN {X 0,Y 752.168,Z 1111.993,A -85,B 0,C 180,E1 34897.654,E2 34897.654} C_VEL
LIN {X 0,Y 752.231,Z 1094.324,A -85,B 0,C 180,E1 34896.499,E2 34896.499} C_VEL
LIN {X 0,Y 752.317,Z 1074.915,A -85,B 0,C 180,E1 34895.381,E2 34895.381} C_VEL
LIN {X 0,Y 752.376,Z 1054.238,A -85,B 0,C 180,E1 34894.368,E2 34894.368} C_VEL
LIN {X 0,Y 752.465,Z 1031.79,A -85,B 0,C 180,E1 34893.439,E2 34893.439} C_VEL
LIN {X 0,Y 752.502,Z 1012.536,A -85,B 0,C 180,E1 34892.77,E2 34892.77} C_VEL
LIN {X 0,Y 752.586,Z 988.881,A -85,B 0,C 180,E1 34892.102,E2 34892.102} C_VEL
LIN {X 0,Y 752.64,Z 966.309,A -85,B 0,C 180,E1 34891.609,E2 34891.609} C_VEL
LIN {X 0,Y 752.681,Z 943.659,A -85,B 0,C 180,E1 34891.263,E2 34891.263} C_VEL
LIN {X 0,Y 752.843,Z 671.726,A -85,B 0,C 180,E1 34888.397,E2 34888.397} C_VEL
LIN {X 0,Y 752.703,Z 602.182,A -85,B 0,C 180,E1 34887.649,E2 34887.649} C_VEL
LIN {X 0,Y 752.426,Z 600.933,A -85,B 0,C 180,E1 34887.619,E2 34887.619} C_VEL
LIN {X 0,Y 752.319,Z 595.825,A -85,B 0,C 180,E1 34887.204,E2 34887.204} C_VEL
LIN {X 0,Y 751.975,Z 594.315,A -85,B 0,C 180,E1 34887.039,E2 34887.039} C_VEL
LIN {X 0,Y 751.973,Z 594.311,A -85,B 0,C 180,E1 34884.075,E2 34884.075} C_VEL
LIN {X 0,Y 751.976,Z 594.309,A -85,B 0,C 180,E1 34881.028,E2 34881.028} C_VEL
LIN {X 0,Y 751.966,Z 594.311,A -85,B 0,C 180,E1 34878.014,E2 34878.014} C_VEL
LIN {X 0,Y 751.991,Z 594.429,A -85,B 0,C 180,E1 34876.965,E2 34876.965} C_VEL
LIN {X 0,Y 751.917,Z 667.686,A -85,B 0,C 180,E1 34874.385,E2 34874.385} C_VEL
LIN {X 0,Y 751.916,Z 711.692,A -85,B 0,C 180,E1 34872.703,E2 34872.703} C_VEL
LIN {X 0,Y 751.921,Z 747.404,A -85,B 0,C 180,E1 34871.217,E2 34871.217} C_VEL
LIN {X 0,Y 752.278,Z 762.857,A -85,B 0,C 180,E1 34870.511,E2 34870.511} C_VEL
LIN {X 0,Y 752.952,Z 773.831,A -85,B 0,C 180,E1 34869.864,E2 34869.864} C_VEL
LIN {X 0,Y 753.854,Z 782.001,A -85,B 0,C 180,E1 34869.231,E2 34869.231} C_VEL
LIN {X 0,Y 754.802,Z 786.816,A -85,B 0,C 180,E1 34868.702,E2 34868.702} C_VEL
LIN {X 0,Y 755.703,Z 789.692,A -85,B 0,C 180,E1 34868.192,E2 34868.192} C_VEL
LIN {X 0,Y 756.47,Z 790.438,A -85,B 0,C 180,E1 34867.734,E2 34867.734} C_VEL
LIN {X 0,Y 756.925,Z 789.304,A -85,B 0,C 180,E1 34867.322,E2 34867.322} C_VEL
LIN {X 0,Y 756.925,Z 786.392,A -85,B 0,C 180,E1 34866.969,E2 34866.969} C_VEL
LIN {X 0,Y 756.484,Z 782.124,A -85,B 0,C 180,E1 34866.717,E2 34866.717} C_VEL
LIN {X 0,Y 755.691,Z 776.229,A -85,B 0,C 180,E1 34866.559,E2 34866.559} C_VEL
LIN {X 0,Y 755.106,Z 767.237,A -85,B 0,C 180,E1 34866.499,E2 34866.499} C_VEL
LIN {X 0,Y 754.991,Z 599.63,A -85,B 0,C 180,E1 34866.488,E2 34866.488} C_VEL
LIN {X 0,Y 752.768,Z 596.94,A -85,B 0,C 180,E1 34866.258,E2 34866.258} C_VEL
LIN {X 0,Y 751.958,Z 594.312,A -85,B 0,C 180,E1 34866.159,E2 34866.159} C_VEL
LIN {X 0,Y 751.987,Z 594.39,A -85,B 0,C 180,E1 34864.473,E2 34864.473} C_VEL
LIN {X 0,Y 752.736,Z 597.93,A -85,B 0,C 180,E1 34864.187,E2 34864.187} C_VEL
LIN {X 0,Y 752.639,Z 638.299,A -85,B 0,C 180,E1 34861.43,E2 34861.43} C_VEL
LIN {X 0,Y 752.635,Z 670.151,A -85,B 0,C 180,E1 34859.331,E2 34859.331} C_VEL
LIN {X 0,Y 752.897,Z 676.713,A -85,B 0,C 180,E1 34859.249,E2 34859.249} C_VEL
LIN {X 0,Y 752.723,Z 950.673,A -85,B 0,C 180,E1 34856.362,E2 34856.362} C_VEL
LIN {X 0,Y 752.667,Z 1018.215,A -85,B 0,C 180,E1 34855.637,E2 34855.637} C_VEL
LIN {X 0,Y 752.631,Z 1041.368,A -85,B 0,C 180,E1 34855.244,E2 34855.244} C_VEL
LIN {X 0,Y 752.572,Z 1063.432,A -85,B 0,C 180,E1 34854.742,E2 34854.742} C_VEL
LIN {X 0,Y 752.514,Z 1085.203,A -85,B 0,C 180,E1 34854.098,E2 34854.098} C_VEL
LIN {X 0,Y 752.449,Z 1106.774,A -85,B 0,C 180,E1 34853.33,E2 34853.33} C_VEL
LIN {X 0,Y 752.37,Z 1127.79,A -85,B 0,C 180,E1 34852.422,E2 34852.422} C_VEL
LIN {X 0,Y 752.284,Z 1148.124,A -85,B 0,C 180,E1 34851.399,E2 34851.399} C_VEL
LIN {X 0,Y 752.226,Z 1166.883,A -85,B 0,C 180,E1 34850.301,E2 34850.301} C_VEL
LIN {X 0,Y 752.154,Z 1185.314,A -85,B 0,C 180,E1 34849.058,E2 34849.058} C_VEL
LIN {X 0,Y 752.099,Z 1202.609,A -85,B 0,C 180,E1 34847.726,E2 34847.726} C_VEL
LIN {X 0,Y 752.048,Z 1218.676,A -85,B 0,C 180,E1 34846.293,E2 34846.293} C_VEL
LIN {X 0,Y 751.998,Z 1233.319,A -85,B 0,C 180,E1 34844.792,E2 34844.792} C_VEL
LIN {X 0,Y 751.97,Z 1246.631,A -85,B 0,C 180,E1 34843.222,E2 34843.222} C_VEL
LIN {X 0,Y 751.948,Z 1258.346,A -85,B 0,C 180,E1 34841.584,E2 34841.584} C_VEL
LIN {X 0,Y 751.924,Z 1268.294,A -85,B 0,C 180,E1 34839.956,E2 34839.956} C_VEL
LIN {X 0,Y 751.921,Z 1276.398,A -85,B 0,C 180,E1 34838.335,E2 34838.335} C_VEL
LIN {X 0,Y 751.899,Z 1283.553,A -85,B 0,C 180,E1 34836.568,E2 34836.568} C_VEL
LIN {X 0,Y 751.904,Z 1288.459,A -85,B 0,C 180,E1 34834.96,E2 34834.96} C_VEL
LIN {X 0,Y 751.912,Z 1292.284,A -85,B 0,C 180,E1 34833.203,E2 34833.203} C_VEL
LIN {X 0,Y 751.891,Z 1294.325,A -85,B 0,C 180,E1 34831.525,E2 34831.525} C_VEL
LIN {X 0,Y 751.895,Z 1294.918,A -85,B 0,C 180,E1 34829.696,E2 34829.696} C_VEL
LIN {X 0,Y 751.913,Z 1293.927,A -85,B 0,C 180,E1 34828.02,E2 34828.02} C_VEL
LIN {X 0,Y 751.897,Z 1291.121,A -85,B 0,C 180,E1 34826.189,E2 34826.189} C_VEL
LIN {X 0,Y 751.899,Z 1287.026,A -85,B 0,C 180,E1 34824.507,E2 34824.507} C_VEL
LIN {X 0,Y 751.924,Z 1280.955,A -85,B 0,C 180,E1 34822.744,E2 34822.744} C_VEL
LIN {X 0,Y 751.913,Z 1273.564,A -85,B 0,C 180,E1 34821.05,E2 34821.05} C_VEL
LIN {X 0,Y 751.928,Z 1264.691,A -85,B 0,C 180,E1 34819.427,E2 34819.427} C_VEL
LIN {X 0,Y 751.951,Z 1254.095,A -85,B 0,C 180,E1 34817.784,E2 34817.784} C_VEL
LIN {X 0,Y 751.983,Z 1242.168,A -85,B 0,C 180,E1 34816.232,E2 34816.232} C_VEL
LIN {X 0,Y 752.016,Z 1228.222,A -85,B 0,C 180,E1 34814.659,E2 34814.659} C_VEL
LIN {X 0,Y 752.06,Z 1212.752,A -85,B 0,C 180,E1 34813.153,E2 34813.153} C_VEL
LIN {X 0,Y 752.11,Z 1196.619,A -85,B 0,C 180,E1 34811.796,E2 34811.796} C_VEL
LIN {X 0,Y 752.181,Z 1178.714,A -85,B 0,C 180,E1 34810.475,E2 34810.475} C_VEL
LIN {X 0,Y 752.236,Z 1160.306,A -85,B 0,C 180,E1 34809.295,E2 34809.295} C_VEL
LIN {X 0,Y 752.324,Z 1140.392,A -85,B 0,C 180,E1 34808.195,E2 34808.195} C_VEL
LIN {X 0,Y 752.402,Z 1120.058,A -85,B 0,C 180,E1 34807.222,E2 34807.222} C_VEL
LIN {X 0,Y 752.47,Z 1099.102,A -85,B 0,C 180,E1 34806.384,E2 34806.384} C_VEL
LIN {X 0,Y 752.545,Z 1077.571,A -85,B 0,C 180,E1 34805.657,E2 34805.657} C_VEL
LIN {X 0,Y 752.58,Z 1055.783,A -85,B 0,C 180,E1 34805.072,E2 34805.072} C_VEL
LIN {X 0,Y 752.653,Z 1032.735,A -85,B 0,C 180,E1 34804.591,E2 34804.591} C_VEL
LIN {X 0,Y 752.67,Z 1011.023,A -85,B 0,C 180,E1 34804.274,E2 34804.274} C_VEL
LIN {X 0,Y 752.868,Z 738.613,A -85,B 0,C 180,E1 34801.41,E2 34801.41} C_VEL
LIN {X 0,Y 752.712,Z 670.505,A -85,B 0,C 180,E1 34800.676,E2 34800.676} C_VEL
LIN {X 0,Y 752.543,Z 668.778,A -85,B 0,C 180,E1 34800.599,E2 34800.599} C_VEL
LIN {X 0,Y 752.672,Z 624.855,A -85,B 0,C 180,E1 34797.661,E2 34797.661} C_VEL
LIN {X 0,Y 752.635,Z 596.643,A -85,B 0,C 180,E1 34795.718,E2 34795.718} C_VEL
LIN {X 0,Y 751.977,Z 594.315,A -85,B 0,C 180,E1 34795.499,E2 34795.499} C_VEL
LIN {X 0,Y 751.994,Z 594.559,A -85,B 0,C 180,E1 34793.822,E2 34793.822} C_VEL
LIN {X 0,Y 753.122,Z 597.562,A -85,B 0,C 180,E1 34793.705,E2 34793.705} C_VEL
LIN {X 0,Y 755.103,Z 599.717,A -85,B 0,C 180,E1 34793.501,E2 34793.501} C_VEL
LIN {X 0,Y 755.254,Z 771.798,A -85,B 0,C 180,E1 34793.485,E2 34793.485} C_VEL
LIN {X 0,Y 756.091,Z 779.16,A -85,B 0,C 180,E1 34793.382,E2 34793.382} C_VEL
LIN {X 0,Y 756.739,Z 784.343,A -85,B 0,C 180,E1 34793.175,E2 34793.175} C_VEL
LIN {X 0,Y 756.992,Z 787.988,A -85,B 0,C 180,E1 34792.871,E2 34792.871} C_VEL
LIN {X 0,Y 756.834,Z 789.825,A -85,B 0,C 180,E1 34792.562,E2 34792.562} C_VEL
LIN {X 0,Y 756.309,Z 790.445,A -85,B 0,C 180,E1 34792.163,E2 34792.163} C_VEL
LIN {X 0,Y 755.519,Z 789.26,A -85,B 0,C 180,E1 34791.703,E2 34791.703} C_VEL
LIN {X 0,Y 754.485,Z 785.515,A -85,B 0,C 180,E1 34791.132,E2 34791.132} C_VEL
LIN {X 0,Y 753.495,Z 779.269,A -85,B 0,C 180,E1 34790.535,E2 34790.535} C_VEL
LIN {X 0,Y 752.759,Z 765.764,A -85,B 0,C 180,E1 34789.563,E2 34789.563} C_VEL
LIN {X 0,Y 752.889,Z 726.4,A -85,B 0,C 180,E1 34786.812,E2 34786.812} C_VEL
LIN {X 0,Y 753.021,Z 688.678,A -85,B 0,C 180,E1 34784.083,E2 34784.083} C_VEL
LIN {X 0,Y 753.149,Z 652.804,A -85,B 0,C 180,E1 34781.388,E2 34781.388} C_VEL
LIN {X 0,Y 753.286,Z 617.67,A -85,B 0,C 180,E1 34778.648,E2 34778.648} C_VEL
LIN {X 0,Y 753.327,Z 597.915,A -85,B 0,C 180,E1 34777.056,E2 34777.056} C_VEL
LIN {X 0,Y 751.956,Z 594.315,A -85,B 0,C 180,E1 34776.633,E2 34776.633} C_VEL
LIN {X 0,Y 751.974,Z 594.315,A -85,B 0,C 180,E1 34773.767,E2 34773.767} C_VEL
LIN {X 0,Y 751.963,Z 594.316,A -85,B 0,C 180,E1 34770.882,E2 34770.882} C_VEL
LIN {X 0,Y 751.95,Z 594.313,A -85,B 0,C 180,E1 34768.081,E2 34768.081} C_VEL
LIN {X 0,Y 751.96,Z 594.311,A -85,B 0,C 180,E1 34765.267,E2 34765.267} C_VEL
LIN {X 0,Y 751.976,Z 594.31,A -85,B 0,C 180,E1 34762.352,E2 34762.352} C_VEL
LIN {X 0,Y 751.971,Z 594.314,A -85,B 0,C 180,E1 34759.416,E2 34759.416} C_VEL
LIN {X 0,Y 751.95,Z 594.316,A -85,B 0,C 180,E1 34756.612,E2 34756.612} C_VEL
LIN {X 0,Y 751.964,Z 594.31,A -85,B 0,C 180,E1 34753.77,E2 34753.77} C_VEL
LIN {X 0,Y 751.973,Z 594.308,A -85,B 0,C 180,E1 34750.884,E2 34750.884} C_VEL
LIN {X 0,Y 751.977,Z 594.308,A -85,B 0,C 180,E1 34747.795,E2 34747.795} C_VEL
LIN {X 0,Y 751.971,Z 594.309,A -85,B 0,C 180,E1 34744.729,E2 34744.729} C_VEL
LIN {X 0,Y 751.974,Z 594.311,A -85,B 0,C 180,E1 34741.753,E2 34741.753} C_VEL
LIN {X 0,Y 751.969,Z 594.316,A -85,B 0,C 180,E1 34738.857,E2 34738.857} C_VEL
LIN {X 0,Y 751.955,Z 594.314,A -85,B 0,C 180,E1 34736.035,E2 34736.035} C_VEL
LIN {X 0,Y 751.966,Z 594.313,A -85,B 0,C 180,E1 34734.428,E2 34734.428} C_VEL
LIN {X 0,Y 750.998,Z 594.439,A -85,B 0,C 180,E1 34733.841,E2 34733.841} C_VEL
LIN {X 0,Y 744.555,Z 595.236,A -85,B 0,C 180,E1 34732.198,E2 34732.198} C_VEL
LIN {X 0,Y 744.013,Z 595.3,A -85,B 0,C 180,E1 34731.771,E2 34731.771} C_VEL
LIN {X 0,Y 744.027,Z 595.3,A -85,B 0,C 180,E1 34728.92,E2 34728.92} C_VEL
LIN {X 0,Y 744.035,Z 595.301,A -85,B 0,C 180,E1 34725.922,E2 34725.922} C_VEL
LIN {X 0,Y 744.039,Z 595.304,A -85,B 0,C 180,E1 34722.964,E2 34722.964} C_VEL
LIN {X 0,Y 744.028,Z 595.303,A -85,B 0,C 180,E1 34720.041,E2 34720.041} C_VEL
LIN {X 0,Y 744.013,Z 595.301,A -85,B 0,C 180,E1 34717.204,E2 34717.204} C_VEL
LIN {X 0,Y 744.028,Z 595.298,A -85,B 0,C 180,E1 34714.359,E2 34714.359} C_VEL
LIN {X 0,Y 744.036,Z 595.298,A -85,B 0,C 180,E1 34711.33,E2 34711.33} C_VEL
LIN {X 0,Y 744.037,Z 595.298,A -85,B 0,C 180,E1 34708.281,E2 34708.281} C_VEL
LIN {X 0,Y 744.03,Z 595.301,A -85,B 0,C 180,E1 34705.263,E2 34705.263} C_VEL
LIN {X 0,Y 744.038,Z 595.304,A -85,B 0,C 180,E1 34702.327,E2 34702.327} C_VEL
LIN {X 0,Y 744.029,Z 595.303,A -85,B 0,C 180,E1 34699.4,E2 34699.4} C_VEL
LIN {X 0,Y 744.017,Z 595.298,A -85,B 0,C 180,E1 34696.521,E2 34696.521} C_VEL
LIN {X 0,Y 744.032,Z 595.298,A -85,B 0,C 180,E1 34693.581,E2 34693.581} C_VEL
LIN {X 0,Y 744.039,Z 595.297,A -85,B 0,C 180,E1 34690.572,E2 34690.572} C_VEL
LIN {X 0,Y 744.036,Z 595.297,A -85,B 0,C 180,E1 34687.499,E2 34687.499} C_VEL
LIN {X 0,Y 744.03,Z 595.299,A -85,B 0,C 180,E1 34684.454,E2 34684.454} C_VEL
LIN {X 0,Y 744.035,Z 595.302,A -85,B 0,C 180,E1 34681.42,E2 34681.42} C_VEL
LIN {X 0,Y 744.057,Z 595.445,A -85,B 0,C 180,E1 34678.58,E2 34678.58} C_VEL
LIN {X 0,Y 745.137,Z 599.811,A -85,B 0,C 180,E1 34678.272,E2 34678.272} C_VEL
LIN {X 0,Y 744.958,Z 645.166,A -85,B 0,C 180,E1 34675.35,E2 34675.35} C_VEL
LIN {X 0,Y 744.723,Z 691.752,A -85,B 0,C 180,E1 34672.413,E2 34672.413} C_VEL
LIN {X 0,Y 744.559,Z 737.788,A -85,B 0,C 180,E1 34669.571,E2 34669.571} C_VEL
LIN {X 0,Y 744.376,Z 785.738,A -85,B 0,C 180,E1 34666.664,E2 34666.664} C_VEL
LIN {X 0,Y 744.3,Z 831.058,A -85,B 0,C 180,E1 34663.978,E2 34663.978} C_VEL
LIN {X 0,Y 744.318,Z 1000.864,A -85,B 0,C 180,E1 34662.302,E2 34662.302} C_VEL
LIN {X 0,Y 744.288,Z 1018.554,A -85,B 0,C 180,E1 34661.978,E2 34661.978} C_VEL
LIN {X 0,Y 744.231,Z 1035.936,A -85,B 0,C 180,E1 34661.507,E2 34661.507} C_VEL
LIN {X 0,Y 744.181,Z 1052.027,A -85,B 0,C 180,E1 34660.919,E2 34660.919} C_VEL
LIN {X 0,Y 744.129,Z 1067.106,A -85,B 0,C 180,E1 34660.215,E2 34660.215} C_VEL
LIN {X 0,Y 744.073,Z 1081.814,A -85,B 0,C 180,E1 34659.357,E2 34659.357} C_VEL
LIN {X 0,Y 744.026,Z 1095.367,A -85,B 0,C 180,E1 34658.383,E2 34658.383} C_VEL
LIN {X 0,Y 743.984,Z 1107.207,A -85,B 0,C 180,E1 34657.334,E2 34657.334} C_VEL
LIN {X 0,Y 743.955,Z 1117.825,A -85,B 0,C 180,E1 34656.171,E2 34656.171} C_VEL
LIN {X 0,Y 743.933,Z 1126.834,A -85,B 0,C 180,E1 34654.934,E2 34654.934} C_VEL
LIN {X 0,Y 743.921,Z 1133.798,A -85,B 0,C 180,E1 34653.698,E2 34653.698} C_VEL
LIN {X 0,Y 743.917,Z 1139.192,A -85,B 0,C 180,E1 34652.387,E2 34652.387} C_VEL
LIN {X 0,Y 743.915,Z 1142.773,A -85,B 0,C 180,E1 34651.077,E2 34651.077} C_VEL
LIN {X 0,Y 743.912,Z 1144.711,A -85,B 0,C 180,E1 34649.691,E2 34649.691} C_VEL
LIN {X 0,Y 743.914,Z 1144.839,A -85,B 0,C 180,E1 34648.382,E2 34648.382} C_VEL
LIN {X 0,Y 743.916,Z 1143.102,A -85,B 0,C 180,E1 34646.994,E2 34646.994} C_VEL
LIN {X 0,Y 743.917,Z 1139.46,A -85,B 0,C 180,E1 34645.605,E2 34645.605} C_VEL
LIN {X 0,Y 743.92,Z 1134.161,A -85,B 0,C 180,E1 34644.291,E2 34644.291} C_VEL
LIN {X 0,Y 743.934,Z 1127.324,A -85,B 0,C 180,E1 34643.051,E2 34643.051} C_VEL
LIN {X 0,Y 743.955,Z 1118.4,A -85,B 0,C 180,E1 34641.808,E2 34641.808} C_VEL
LIN {X 0,Y 743.98,Z 1107.845,A -85,B 0,C 180,E1 34640.64,E2 34640.64} C_VEL
LIN {X 0,Y 744.019,Z 1096.581,A -85,B 0,C 180,E1 34639.624,E2 34639.624} C_VEL
LIN {X 0,Y 744.068,Z 1083.83,A -85,B 0,C 180,E1 34638.684,E2 34638.684} C_VEL
LIN {X 0,Y 744.12,Z 1069.433,A -85,B 0,C 180,E1 34637.82,E2 34637.82} C_VEL
LIN {X 0,Y 744.168,Z 1053.947,A -85,B 0,C 180,E1 34637.072,E2 34637.072} C_VEL
LIN {X 0,Y 744.223,Z 1038.349,A -85,B 0,C 180,E1 34636.48,E2 34636.48} C_VEL
LIN {X 0,Y 744.284,Z 1021.006,A -85,B 0,C 180,E1 34635.988,E2 34635.988} C_VEL
LIN {X 0,Y 744.315,Z 1003.236,A -85,B 0,C 180,E1 34635.644,E2 34635.644} C_VEL
LIN {X 0,Y 744.341,Z 976.491,A -85,B 0,C 180,E1 34635.351,E2 34635.351} C_VEL
LIN {X 0,Y 744.254,Z 830.555,A -85,B 0,C 180,E1 34633.922,E2 34633.922} C_VEL
LIN {X 0,Y 744.405,Z 780.799,A -85,B 0,C 180,E1 34630.949,E2 34630.949} C_VEL
LIN {X 0,Y 744.581,Z 730.791,A -85,B 0,C 180,E1 34627.911,E2 34627.911} C_VEL
LIN {X 0,Y 744.743,Z 685.834,A -85,B 0,C 180,E1 34625.127,E2 34625.127} C_VEL
LIN {X 0,Y 744.951,Z 642.027,A -85,B 0,C 180,E1 34622.359,E2 34622.359} C_VEL
LIN {X 0,Y 745.136,Z 599.341,A -85,B 0,C 180,E1 34619.609,E2 34619.609} C_VEL
LIN {X 0,Y 744.012,Z 595.307,A -85,B 0,C 180,E1 34619.31,E2 34619.31} C_VEL
LIN {X 0,Y 744.02,Z 595.296,A -85,B 0,C 180,E1 34616.471,E2 34616.471} C_VEL
LIN {X 0,Y 744.034,Z 595.296,A -85,B 0,C 180,E1 34613.609,E2 34613.609} C_VEL
LIN {X 0,Y 744.037,Z 595.292,A -85,B 0,C 180,E1 34610.531,E2 34610.531} C_VEL
LIN {X 0,Y 744.017,Z 595.299,A -85,B 0,C 180,E1 34607.659,E2 34607.659} C_VEL
LIN {X 0,Y 744.015,Z 595.301,A -85,B 0,C 180,E1 34604.875,E2 34604.875} C_VEL
LIN {X 0,Y 744.032,Z 595.294,A -85,B 0,C 180,E1 34601.998,E2 34601.998} C_VEL
LIN {X 0,Y 744.037,Z 595.298,A -85,B 0,C 180,E1 34598.972,E2 34598.972} C_VEL
LIN {X 0,Y 744.026,Z 595.296,A -85,B 0,C 180,E1 34596.06,E2 34596.06} C_VEL
LIN {X 0,Y 744.016,Z 595.304,A -85,B 0,C 180,E1 34593.148,E2 34593.148} C_VEL
LIN {X 0,Y 744.015,Z 595.297,A -85,B 0,C 180,E1 34590.352,E2 34590.352} C_VEL
LIN {X 0,Y 744.029,Z 595.306,A -85,B 0,C 180,E1 34587.449,E2 34587.449} C_VEL
LIN {X 0,Y 744.03,Z 595.443,A -85,B 0,C 180,E1 34587.102,E2 34587.102} C_VEL
LIN {X 0,Y 745,Z 600.148,A -85,B 0,C 180,E1 34586.676,E2 34586.676} C_VEL
LIN {X 0,Y 745.112,Z 601.561,A -85,B 0,C 180,E1 34586.596,E2 34586.596} C_VEL
LIN {X 0,Y 745.899,Z 605.701,A -85,B 0,C 180,E1 34586.517,E2 34586.517} C_VEL
LIN {X 0,Y 745.576,Z 863.201,A -85,B 0,C 180,E1 34583.774,E2 34583.774} C_VEL
LIN {X 0,Y 745.454,Z 947.006,A -85,B 0,C 180,E1 34582.873,E2 34582.873} C_VEL
LIN {X 0,Y 745.359,Z 970.922,A -85,B 0,C 180,E1 34582.472,E2 34582.472} C_VEL
LIN {X 0,Y 745.257,Z 993.169,A -85,B 0,C 180,E1 34581.962,E2 34581.962} C_VEL
LIN {X 0,Y 745.107,Z 1014.667,A -85,B 0,C 180,E1 34581.326,E2 34581.326} C_VEL
LIN {X 0,Y 745.004,Z 1036.415,A -85,B 0,C 180,E1 34580.547,E2 34580.547} C_VEL
LIN {X 0,Y 744.837,Z 1057.946,A -85,B 0,C 180,E1 34579.61,E2 34579.61} C_VEL
LIN {X 0,Y 744.667,Z 1078.632,A -85,B 0,C 180,E1 34578.556,E2 34578.556} C_VEL
LIN {X 0,Y 744.545,Z 1098.247,A -85,B 0,C 180,E1 34577.389,E2 34577.389} C_VEL
LIN {X 0,Y 744.392,Z 1116.888,A -85,B 0,C 180,E1 34576.104,E2 34576.104} C_VEL
LIN {X 0,Y 744.274,Z 1133.588,A -85,B 0,C 180,E1 34574.789,E2 34574.789} C_VEL
LIN {X 0,Y 744.181,Z 1149.333,A -85,B 0,C 180,E1 34573.362,E2 34573.362} C_VEL
LIN {X 0,Y 744.086,Z 1164.405,A -85,B 0,C 180,E1 34571.786,E2 34571.786} C_VEL
LIN {X 0,Y 744.017,Z 1177.399,A -85,B 0,C 180,E1 34570.218,E2 34570.218} C_VEL
LIN {X 0,Y 743.975,Z 1188.389,A -85,B 0,C 180,E1 34568.657,E2 34568.657} C_VEL
LIN {X 0,Y 743.952,Z 1198.665,A -85,B 0,C 180,E1 34566.948,E2 34566.948} C_VEL
LIN {X 0,Y 743.927,Z 1207.025,A -85,B 0,C 180,E1 34565.244,E2 34565.244} C_VEL
LIN {X 0,Y 743.908,Z 1214.22,A -85,B 0,C 180,E1 34563.391,E2 34563.391} C_VEL
LIN {X 0,Y 743.903,Z 1218.974,A -85,B 0,C 180,E1 34561.772,E2 34561.772} C_VEL
LIN {X 0,Y 743.91,Z 1222.678,A -85,B 0,C 180,E1 34559.923,E2 34559.923} C_VEL
LIN {X 0,Y 743.914,Z 1224.627,A -85,B 0,C 180,E1 34558.151,E2 34558.151} C_VEL
LIN {X 0,Y 743.917,Z 1224.837,A -85,B 0,C 180,E1 34556.378,E2 34556.378} C_VEL
LIN {X 0,Y 743.909,Z 1223.571,A -85,B 0,C 180,E1 34554.601,E2 34554.601} C_VEL
LIN {X 0,Y 743.915,Z 1220.544,A -85,B 0,C 180,E1 34552.819,E2 34552.819} C_VEL
LIN {X 0,Y 743.913,Z 1215.63,A -85,B 0,C 180,E1 34550.952,E2 34550.952} C_VEL
LIN {X 0,Y 743.908,Z 1210.056,A -85,B 0,C 180,E1 34549.389,E2 34549.389} C_VEL
LIN {X 0,Y 743.934,Z 1201.894,A -85,B 0,C 180,E1 34547.582,E2 34547.582} C_VEL
LIN {X 0,Y 743.969,Z 1192.65,A -85,B 0,C 180,E1 34545.921,E2 34545.921} C_VEL
LIN {X 0,Y 744,Z 1181.195,A -85,B 0,C 180,E1 34544.21,E2 34544.21} C_VEL
LIN {X 0,Y 744.069,Z 1168.962,A -85,B 0,C 180,E1 34542.643,E2 34542.643} C_VEL
LIN {X 0,Y 744.129,Z 1154.907,A -85,B 0,C 180,E1 34541.105,E2 34541.105} C_VEL
LIN {X 0,Y 744.249,Z 1138.569,A -85,B 0,C 180,E1 34539.555,E2 34539.555} C_VEL
LIN {X 0,Y 744.355,Z 1122.079,A -85,B 0,C 180,E1 34538.192,E2 34538.192} C_VEL
LIN {X 0,Y 744.472,Z 1104.145,A -85,B 0,C 180,E1 34536.91,E2 34536.91} C_VEL
LIN {X 0,Y 744.638,Z 1083.916,A -85,B 0,C 180,E1 34535.655,E2 34535.655} C_VEL
LIN {X 0,Y 744.784,Z 1064.229,A -85,B 0,C 180,E1 34534.6,E2 34534.6} C_VEL
LIN {X 0,Y 744.936,Z 1043.678,A -85,B 0,C 180,E1 34533.665,E2 34533.665} C_VEL
LIN {X 0,Y 745.088,Z 1021.603,A -85,B 0,C 180,E1 34532.814,E2 34532.814} C_VEL
LIN {X 0,Y 745.206,Z 1000.64,A -85,B 0,C 180,E1 34532.157,E2 34532.157} C_VEL
LIN {X 0,Y 745.33,Z 977.796,A -85,B 0,C 180,E1 34531.578,E2 34531.578} C_VEL
LIN {X 0,Y 745.423,Z 955.321,A -85,B 0,C 180,E1 34531.159,E2 34531.159} C_VEL
LIN {X 0,Y 745.499,Z 925.596,A -85,B 0,C 180,E1 34530.791,E2 34530.791} C_VEL
LIN {X 0,Y 745.826,Z 664.126,A -85,B 0,C 180,E1 34528.022,E2 34528.022} C_VEL
LIN {X 0,Y 745.725,Z 603.799,A -85,B 0,C 180,E1 34527.365,E2 34527.365} C_VEL
LIN {X 0,Y 744.983,Z 600.806,A -85,B 0,C 180,E1 34527.287,E2 34527.287} C_VEL
LIN {X 0,Y 744.582,Z 597.37,A -85,B 0,C 180,E1 34526.99,E2 34526.99} C_VEL
LIN {X 0,Y 744.032,Z 595.306,A -85,B 0,C 180,E1 34526.795,E2 34526.795} C_VEL
LIN {X 0,Y 744.022,Z 595.304,A -85,B 0,C 180,E1 34523.871,E2 34523.871} C_VEL
LIN {X 0,Y 744.038,Z 595.3,A -85,B 0,C 180,E1 34520.929,E2 34520.929} C_VEL
LIN {X 0,Y 744.036,Z 595.3,A -85,B 0,C 180,E1 34517.887,E2 34517.887} C_VEL
LIN {X 0,Y 744.044,Z 595.34,A -85,B 0,C 180,E1 34517.098,E2 34517.098} C_VEL
LIN {X 0,Y 743.982,Z 615.25,A -85,B 0,C 180,E1 34516.306,E2 34516.306} C_VEL
LIN {X 0,Y 743.921,Z 679.905,A -85,B 0,C 180,E1 34513.947,E2 34513.947} C_VEL
LIN {X 0,Y 743.92,Z 725.916,A -85,B 0,C 180,E1 34512.122,E2 34512.122} C_VEL
LIN {X 0,Y 744.482,Z 766.921,A -85,B 0,C 180,E1 34510.369,E2 34510.369} C_VEL
LIN {X 0,Y 745.666,Z 778.687,A -85,B 0,C 180,E1 34509.793,E2 34509.793} C_VEL
LIN {X 0,Y 747.168,Z 786.751,A -85,B 0,C 180,E1 34509.272,E2 34509.272} C_VEL
LIN {X 0,Y 749.097,Z 792.682,A -85,B 0,C 180,E1 34508.728,E2 34508.728} C_VEL
LIN {X 0,Y 750.911,Z 796.108,A -85,B 0,C 180,E1 34508.221,E2 34508.221} C_VEL
LIN {X 0,Y 752.462,Z 797.41,A -85,B 0,C 180,E1 34507.753,E2 34507.753} C_VEL
LIN {X 0,Y 753.548,Z 796.999,A -85,B 0,C 180,E1 34507.33,E2 34507.33} C_VEL
LIN {X 0,Y 754.077,Z 794.942,A -85,B 0,C 180,E1 34506.911,E2 34506.911} C_VEL
LIN {X 0,Y 753.83,Z 791.367,A -85,B 0,C 180,E1 34506.553,E2 34506.553} C_VEL
LIN {X 0,Y 752.837,Z 786.449,A -85,B 0,C 180,E1 34506.284,E2 34506.284} C_VEL
LIN {X 0,Y 751.257,Z 779.244,A -85,B 0,C 180,E1 34506.101,E2 34506.101} C_VEL
LIN {X 0,Y 750.428,Z 770.079,A -85,B 0,C 180,E1 34506.014,E2 34506.014} C_VEL
LIN {X 0,Y 750.262,Z 603.955,A -85,B 0,C 180,E1 34505.997,E2 34505.997} C_VEL
LIN {X 0,Y 748.796,Z 601.662,A -85,B 0,C 180,E1 34505.842,E2 34505.842} C_VEL
LIN {X 0,Y 745.88,Z 599.501,A -85,B 0,C 180,E1 34505.531,E2 34505.531} C_VEL
LIN {X 0,Y 744.321,Z 596.634,A -85,B 0,C 180,E1 34505.362,E2 34505.362} C_VEL
LIN {X 0,Y 744.036,Z 595.298,A -85,B 0,C 180,E1 34505.325,E2 34505.325} C_VEL
LIN {X 0,Y 744.042,Z 595.408,A -85,B 0,C 180,E1 34504.822,E2 34504.822} C_VEL
LIN {X 0,Y 745.588,Z 600.578,A -85,B 0,C 180,E1 34504.375,E2 34504.375} C_VEL
LIN {X 0,Y 745.365,Z 641.006,A -85,B 0,C 180,E1 34501.587,E2 34501.587} C_VEL
LIN {X 0,Y 745.267,Z 670.1,A -85,B 0,C 180,E1 34499.65,E2 34499.65} C_VEL
LIN {X 0,Y 745.917,Z 674.305,A -85,B 0,C 180,E1 34499.576,E2 34499.576} C_VEL
LIN {X 0,Y 745.551,Z 950.164,A -85,B 0,C 180,E1 34496.641,E2 34496.641} C_VEL
LIN {X 0,Y 745.448,Z 1018.454,A -85,B 0,C 180,E1 34495.901,E2 34495.901} C_VEL
LIN {X 0,Y 745.36,Z 1041.75,A -85,B 0,C 180,E1 34495.5,E2 34495.5} C_VEL
LIN {X 0,Y 745.255,Z 1063.436,A -85,B 0,C 180,E1 34495.001,E2 34495.001} C_VEL
LIN {X 0,Y 745.123,Z 1085.932,A -85,B 0,C 180,E1 34494.329,E2 34494.329} C_VEL
LIN {X 0,Y 744.986,Z 1107.401,A -85,B 0,C 180,E1 34493.552,E2 34493.552} C_VEL
LIN {X 0,Y 744.835,Z 1127.8,A -85,B 0,C 180,E1 34492.662,E2 34492.662} C_VEL
LIN {X 0,Y 744.661,Z 1148.854,A -85,B 0,C 180,E1 34491.588,E2 34491.588} C_VEL
LIN {X 0,Y 744.541,Z 1168.211,A -85,B 0,C 180,E1 34490.437,E2 34490.437} C_VEL
LIN {X 0,Y 744.394,Z 1186.552,A -85,B 0,C 180,E1 34489.174,E2 34489.174} C_VEL
LIN {X 0,Y 744.265,Z 1204.466,A -85,B 0,C 180,E1 34487.757,E2 34487.757} C_VEL
LIN {X 0,Y 744.18,Z 1220.369,A -85,B 0,C 180,E1 34486.31,E2 34486.31} C_VEL
LIN {X 0,Y 744.086,Z 1234.734,A -85,B 0,C 180,E1 34484.793,E2 34484.793} C_VEL
LIN {X 0,Y 744.021,Z 1247.812,A -85,B 0,C 180,E1 34483.207,E2 34483.207} C_VEL
LIN {X 0,Y 743.983,Z 1258.868,A -85,B 0,C 180,E1 34481.631,E2 34481.631} C_VEL
LIN {X 0,Y 743.936,Z 1269.519,A -85,B 0,C 180,E1 34479.829,E2 34479.829} C_VEL
LIN {X 0,Y 743.932,Z 1277.463,A -85,B 0,C 180,E1 34478.192,E2 34478.192} C_VEL
LIN {X 0,Y 743.911,Z 1284.315,A -85,B 0,C 180,E1 34476.406,E2 34476.406} C_VEL
LIN {X 0,Y 743.895,Z 1289.077,A -85,B 0,C 180,E1 34474.781,E2 34474.781} C_VEL
LIN {X 0,Y 743.906,Z 1292.736,A -85,B 0,C 180,E1 34472.929,E2 34472.929} C_VEL
LIN {X 0,Y 743.907,Z 1294.657,A -85,B 0,C 180,E1 34471.156,E2 34471.156} C_VEL
LIN {X 0,Y 743.891,Z 1294.852,A -85,B 0,C 180,E1 34469.462,E2 34469.462} C_VEL
LIN {X 0,Y 743.9,Z 1293.629,A -85,B 0,C 180,E1 34467.69,E2 34467.69} C_VEL
LIN {X 0,Y 743.913,Z 1290.65,A -85,B 0,C 180,E1 34465.916,E2 34465.916} C_VEL
LIN {X 0,Y 743.906,Z 1285.839,A -85,B 0,C 180,E1 34464.061,E2 34464.061} C_VEL
LIN {X 0,Y 743.911,Z 1280.047,A -85,B 0,C 180,E1 34462.432,E2 34462.432} C_VEL
LIN {X 0,Y 743.947,Z 1271.972,A -85,B 0,C 180,E1 34460.642,E2 34460.642} C_VEL
LIN {X 0,Y 743.959,Z 1262.849,A -85,B 0,C 180,E1 34458.999,E2 34458.999} C_VEL
LIN {X 0,Y 744.003,Z 1251.842,A -85,B 0,C 180,E1 34457.343,E2 34457.343} C_VEL
LIN {X 0,Y 744.047,Z 1240.247,A -85,B 0,C 180,E1 34455.844,E2 34455.844} C_VEL
LIN {X 0,Y 744.139,Z 1225.9,A -85,B 0,C 180,E1 34454.252,E2 34454.252} C_VEL
LIN {X 0,Y 744.233,Z 1210.794,A -85,B 0,C 180,E1 34452.794,E2 34452.794} C_VEL
LIN {X 0,Y 744.327,Z 1194.594,A -85,B 0,C 180,E1 34451.437,E2 34451.437} C_VEL
LIN {X 0,Y 744.469,Z 1176.84,A -85,B 0,C 180,E1 34450.137,E2 34450.137} C_VEL
LIN {X 0,Y 744.618,Z 1158.302,A -85,B 0,C 180,E1 34448.95,E2 34448.95} C_VEL
LIN {X 0,Y 744.752,Z 1137.993,A -85,B 0,C 180,E1 34447.837,E2 34447.837} C_VEL
LIN {X 0,Y 744.926,Z 1116.059,A -85,B 0,C 180,E1 34446.811,E2 34446.811} C_VEL
LIN {X 0,Y 745.043,Z 1095.756,A -85,B 0,C 180,E1 34446.007,E2 34446.007} C_VEL
LIN {X 0,Y 745.203,Z 1073.462,A -85,B 0,C 180,E1 34445.283,E2 34445.283} C_VEL
LIN {X 0,Y 745.293,Z 1052.089,A -85,B 0,C 180,E1 34444.72,E2 34444.72} C_VEL
LIN {X 0,Y 745.413,Z 1028.86,A -85,B 0,C 180,E1 34444.262,E2 34444.262} C_VEL
LIN {X 0,Y 745.465,Z 1006.354,A -85,B 0,C 180,E1 34443.948,E2 34443.948} C_VEL
LIN {X 0,Y 745.832,Z 743.748,A -85,B 0,C 180,E1 34441.17,E2 34441.17} C_VEL
LIN {X 0,Y 745.744,Z 672.096,A -85,B 0,C 180,E1 34440.392,E2 34440.392} C_VEL
LIN {X 0,Y 745.188,Z 669.44,A -85,B 0,C 180,E1 34440.324,E2 34440.324} C_VEL
LIN {X 0,Y 745.453,Z 626.016,A -85,B 0,C 180,E1 34437.389,E2 34437.389} C_VEL
LIN {X 0,Y 745.501,Z 599.922,A -85,B 0,C 180,E1 34435.575,E2 34435.575} C_VEL
LIN {X 0,Y 744.023,Z 595.307,A -85,B 0,C 180,E1 34435.148,E2 34435.148} C_VEL
LIN {X 0,Y 744.071,Z 595.536,A -85,B 0,C 180,E1 34434.665,E2 34434.665} C_VEL
LIN {X 0,Y 745.139,Z 598.469,A -85,B 0,C 180,E1 34434.549,E2 34434.549} C_VEL
LIN {X 0,Y 747.611,Z 601.029,A -85,B 0,C 180,E1 34434.284,E2 34434.284} C_VEL
LIN {X 0,Y 749.147,Z 602.056,A -85,B 0,C 180,E1 34434.121,E2 34434.121} C_VEL
LIN {X 0,Y 750.371,Z 604.11,A -85,B 0,C 180,E1 34433.992,E2 34433.992} C_VEL
LIN {X 0,Y 750.522,Z 772.222,A -85,B 0,C 180,E1 34433.976,E2 34433.976} C_VEL
LIN {X 0,Y 751.534,Z 780.853,A -85,B 0,C 180,E1 34433.87,E2 34433.87} C_VEL
LIN {X 0,Y 753.029,Z 787.264,A -85,B 0,C 180,E1 34433.682,E2 34433.682} C_VEL
LIN {X 0,Y 753.919,Z 792.036,A -85,B 0,C 180,E1 34433.395,E2 34433.395} C_VEL
LIN {X 0,Y 754.045,Z 795.328,A -85,B 0,C 180,E1 34433.035,E2 34433.035} C_VEL
LIN {X 0,Y 753.495,Z 797.068,A -85,B 0,C 180,E1 34432.644,E2 34432.644} C_VEL
LIN {X 0,Y 752.381,Z 797.385,A -85,B 0,C 180,E1 34432.22,E2 34432.22} C_VEL
LIN {X 0,Y 750.755,Z 795.908,A -85,B 0,C 180,E1 34431.736,E2 34431.736} C_VEL
LIN {X 0,Y 748.952,Z 792.312,A -85,B 0,C 180,E1 34431.231,E2 34431.231} C_VEL
LIN {X 0,Y 747.055,Z 786.197,A -85,B 0,C 180,E1 34430.68,E2 34430.68} C_VEL
LIN {X 0,Y 745.699,Z 774.283,A -85,B 0,C 180,E1 34429.789,E2 34429.789} C_VEL
LIN {X 0,Y 745.869,Z 729.073,A -85,B 0,C 180,E1 34426.602,E2 34426.602} C_VEL
LIN {X 0,Y 746.139,Z 691.45,A -85,B 0,C 180,E1 34423.854,E2 34423.854} C_VEL
LIN {X 0,Y 746.404,Z 655.957,A -85,B 0,C 180,E1 34421.164,E2 34421.164} C_VEL
LIN {X 0,Y 746.668,Z 620.984,A -85,B 0,C 180,E1 34418.416,E2 34418.416} C_VEL
LIN {X 0,Y 746.629,Z 601.972,A -85,B 0,C 180,E1 34416.868,E2 34416.868} C_VEL
LIN {X 0,Y 744.037,Z 595.422,A -85,B 0,C 180,E1 34416.122,E2 34416.122} C_VEL
LIN {X 0,Y 744.012,Z 595.301,A -85,B 0,C 180,E1 34413.252,E2 34413.252} C_VEL
LIN {X 0,Y 744.019,Z 595.304,A -85,B 0,C 180,E1 34410.441,E2 34410.441} C_VEL
LIN {X 0,Y 744.038,Z 595.304,A -85,B 0,C 180,E1 34407.535,E2 34407.535} C_VEL
LIN {X 0,Y 744.026,Z 595.303,A -85,B 0,C 180,E1 34404.621,E2 34404.621} C_VEL
LIN {X 0,Y 744.012,Z 595.301,A -85,B 0,C 180,E1 34401.773,E2 34401.773} C_VEL
LIN {X 0,Y 744.019,Z 595.3,A -85,B 0,C 180,E1 34398.979,E2 34398.979} C_VEL
LIN {X 0,Y 744.034,Z 595.301,A -85,B 0,C 180,E1 34396.072,E2 34396.072} C_VEL
LIN {X 0,Y 744.034,Z 595.304,A -85,B 0,C 180,E1 34393.127,E2 34393.127} C_VEL
LIN {X 0,Y 744.015,Z 595.303,A -85,B 0,C 180,E1 34390.296,E2 34390.296} C_VEL
LIN {X 0,Y 744.019,Z 595.3,A -85,B 0,C 180,E1 34387.49,E2 34387.49} C_VEL
LIN {X 0,Y 744.028,Z 595.298,A -85,B 0,C 180,E1 34384.548,E2 34384.548} C_VEL
LIN {X 0,Y 744.035,Z 595.297,A -85,B 0,C 180,E1 34381.54,E2 34381.54} C_VEL
LIN {X 0,Y 744.033,Z 595.298,A -85,B 0,C 180,E1 34378.46,E2 34378.46} C_VEL
LIN {X 0,Y 744.038,Z 595.3,A -85,B 0,C 180,E1 34375.452,E2 34375.452} C_VEL
LIN {X 0,Y 744.035,Z 595.305,A -85,B 0,C 180,E1 34372.51,E2 34372.51} C_VEL
LIN {X 0,Y 744.013,Z 595.3,A -85,B 0,C 180,E1 34371.771,E2 34371.771} C_VEL
LIN {X 0,Y 743.024,Z 595.429,A -85,B 0,C 180,E1 34371.178,E2 34371.178} C_VEL
LIN {X 0,Y 736.636,Z 596.226,A -85,B 0,C 180,E1 34369.516,E2 34369.516} C_VEL
LIN {X 0,Y 736.098,Z 596.289,A -85,B 0,C 180,E1 34369.084,E2 34369.084} C_VEL
LIN {X 0,Y 736.098,Z 596.292,A -85,B 0,C 180,E1 34366.088,E2 34366.088} C_VEL
LIN {X 0,Y 736.081,Z 596.293,A -85,B 0,C 180,E1 34363.182,E2 34363.182} C_VEL
LIN {X 0,Y 736.081,Z 596.289,A -85,B 0,C 180,E1 34360.313,E2 34360.313} C_VEL
LIN {X 0,Y 736.089,Z 596.287,A -85,B 0,C 180,E1 34357.468,E2 34357.468} C_VEL
LIN {X 0,Y 736.095,Z 596.287,A -85,B 0,C 180,E1 34354.494,E2 34354.494} C_VEL
LIN {X 0,Y 736.096,Z 596.288,A -85,B 0,C 180,E1 34351.435,E2 34351.435} C_VEL
LIN {X 0,Y 736.098,Z 596.288,A -85,B 0,C 180,E1 34348.377,E2 34348.377} C_VEL
LIN {X 0,Y 736.087,Z 596.292,A -85,B 0,C 180,E1 34345.402,E2 34345.402} C_VEL
LIN {X 0,Y 736.076,Z 596.293,A -85,B 0,C 180,E1 34342.612,E2 34342.612} C_VEL
LIN {X 0,Y 736.089,Z 596.288,A -85,B 0,C 180,E1 34339.715,E2 34339.715} C_VEL
LIN {X 0,Y 736.091,Z 596.283,A -85,B 0,C 180,E1 34336.724,E2 34336.724} C_VEL
LIN {X 0,Y 736.098,Z 596.286,A -85,B 0,C 180,E1 34333.726,E2 34333.726} C_VEL
LIN {X 0,Y 736.091,Z 596.288,A -85,B 0,C 180,E1 34330.692,E2 34330.692} C_VEL
LIN {X 0,Y 736.093,Z 596.289,A -85,B 0,C 180,E1 34327.76,E2 34327.76} C_VEL
LIN {X 0,Y 736.095,Z 596.293,A -85,B 0,C 180,E1 34324.869,E2 34324.869} C_VEL
LIN {X 0,Y 736.081,Z 596.293,A -85,B 0,C 180,E1 34321.988,E2 34321.988} C_VEL
LIN {X 0,Y 736.099,Z 596.29,A -85,B 0,C 180,E1 34319.007,E2 34319.007} C_VEL
LIN {X 0,Y 736.124,Z 596.502,A -85,B 0,C 180,E1 34318.783,E2 34318.783} C_VEL
LIN {X 0,Y 737.555,Z 602.195,A -85,B 0,C 180,E1 34318.377,E2 34318.377} C_VEL
LIN {X 0,Y 737.558,Z 634.728,A -85,B 0,C 180,E1 34316.313,E2 34316.313} C_VEL
LIN {X 0,Y 737.248,Z 680.701,A -85,B 0,C 180,E1 34313.366,E2 34313.366} C_VEL
LIN {X 0,Y 736.937,Z 726.591,A -85,B 0,C 180,E1 34310.489,E2 34310.489} C_VEL
LIN {X 0,Y 736.702,Z 772.311,A -85,B 0,C 180,E1 34307.675,E2 34307.675} C_VEL
LIN {X 0,Y 736.475,Z 820.644,A -85,B 0,C 180,E1 34304.746,E2 34304.746} C_VEL
LIN {X 0,Y 736.471,Z 831.016,A -85,B 0,C 180,E1 34304.142,E2 34304.142} C_VEL
LIN {X 0,Y 736.618,Z 902.094,A -85,B 0,C 180,E1 34303.437,E2 34303.437} C_VEL
LIN {X 0,Y 736.528,Z 1001.151,A -85,B 0,C 180,E1 34302.442,E2 34302.442} C_VEL
LIN {X 0,Y 736.48,Z 1018.961,A -85,B 0,C 180,E1 34302.109,E2 34302.109} C_VEL
LIN {X 0,Y 736.398,Z 1036.308,A -85,B 0,C 180,E1 34301.631,E2 34301.631} C_VEL
LIN {X 0,Y 736.322,Z 1052.305,A -85,B 0,C 180,E1 34301.037,E2 34301.037} C_VEL
LIN {X 0,Y 736.239,Z 1067.321,A -85,B 0,C 180,E1 34300.326,E2 34300.326} C_VEL
LIN {X 0,Y 736.152,Z 1081.993,A -85,B 0,C 180,E1 34299.458,E2 34299.458} C_VEL
LIN {X 0,Y 736.082,Z 1095.509,A -85,B 0,C 180,E1 34298.474,E2 34298.474} C_VEL
LIN {X 0,Y 736.019,Z 1107.323,A -85,B 0,C 180,E1 34297.414,E2 34297.414} C_VEL
LIN {X 0,Y 735.974,Z 1117.921,A -85,B 0,C 180,E1 34296.239,E2 34296.239} C_VEL
LIN {X 0,Y 735.942,Z 1126.906,A -85,B 0,C 180,E1 34294.987,E2 34294.987} C_VEL
LIN {X 0,Y 735.925,Z 1133.852,A -85,B 0,C 180,E1 34293.738,E2 34293.738} C_VEL
LIN {X 0,Y 735.919,Z 1139.229,A -85,B 0,C 180,E1 34292.413,E2 34292.413} C_VEL
LIN {X 0,Y 735.917,Z 1142.953,A -85,B 0,C 180,E1 34291.011,E2 34291.011} C_VEL
LIN {X 0,Y 735.913,Z 1144.787,A -85,B 0,C 180,E1 34289.61,E2 34289.61} C_VEL
LIN {X 0,Y 735.913,Z 1144.775,A -85,B 0,C 180,E1 34288.286,E2 34288.286} C_VEL
LIN {X 0,Y 735.917,Z 1142.923,A -85,B 0,C 180,E1 34286.884,E2 34286.884} C_VEL
LIN {X 0,Y 735.918,Z 1139.424,A -85,B 0,C 180,E1 34285.557,E2 34285.557} C_VEL
LIN {X 0,Y 735.924,Z 1134.11,A -85,B 0,C 180,E1 34284.229,E2 34284.229} C_VEL
LIN {X 0,Y 735.943,Z 1127.248,A -85,B 0,C 180,E1 34282.975,E2 34282.975} C_VEL
LIN {X 0,Y 735.974,Z 1118.308,A -85,B 0,C 180,E1 34281.719,E2 34281.719} C_VEL
LIN {X 0,Y 736.014,Z 1107.734,A -85,B 0,C 180,E1 34280.538,E2 34280.538} C_VEL
LIN {X 0,Y 736.076,Z 1096.447,A -85,B 0,C 180,E1 34279.511,E2 34279.511} C_VEL
LIN {X 0,Y 736.15,Z 1083.053,A -85,B 0,C 180,E1 34278.521,E2 34278.521} C_VEL
LIN {X 0,Y 736.23,Z 1068.492,A -85,B 0,C 180,E1 34277.648,E2 34277.648} C_VEL
LIN {X 0,Y 736.308,Z 1053.677,A -85,B 0,C 180,E1 34276.931,E2 34276.931} C_VEL
LIN {X 0,Y 736.39,Z 1037.986,A -85,B 0,C 180,E1 34276.333,E2 34276.333} C_VEL
LIN {X 0,Y 736.478,Z 1020.508,A -85,B 0,C 180,E1 34275.836,E2 34275.836} C_VEL
LIN {X 0,Y 736.526,Z 1002.457,A -85,B 0,C 180,E1 34275.488,E2 34275.488} C_VEL
LIN {X 0,Y 736.575,Z 969.575,A -85,B 0,C 180,E1 34275.137,E2 34275.137} C_VEL
LIN {X 0,Y 736.473,Z 831.001,A -85,B 0,C 180,E1 34273.768,E2 34273.768} C_VEL
LIN {X 0,Y 736.658,Z 782.525,A -85,B 0,C 180,E1 34270.858,E2 34270.858} C_VEL
LIN {X 0,Y 736.919,Z 732.646,A -85,B 0,C 180,E1 34267.797,E2 34267.797} C_VEL
LIN {X 0,Y 737.178,Z 687.348,A -85,B 0,C 180,E1 34264.963,E2 34264.963} C_VEL
LIN {X 0,Y 737.486,Z 644.033,A -85,B 0,C 180,E1 34262.199,E2 34262.199} C_VEL
LIN {X 0,Y 737.596,Z 612.237,A -85,B 0,C 180,E1 34260.164,E2 34260.164} C_VEL
LIN {X 0,Y 737.289,Z 600.674,A -85,B 0,C 180,E1 34259.431,E2 34259.431} C_VEL
LIN {X 0,Y 736.084,Z 596.296,A -85,B 0,C 180,E1 34259.104,E2 34259.104} C_VEL
LIN {X 0,Y 736.073,Z 596.284,A -85,B 0,C 180,E1 34256.238,E2 34256.238} C_VEL
LIN {X 0,Y 736.086,Z 596.29,A -85,B 0,C 180,E1 34253.392,E2 34253.392} C_VEL
LIN {X 0,Y 736.097,Z 596.28,A -85,B 0,C 180,E1 34250.425,E2 34250.425} C_VEL
LIN {X 0,Y 736.092,Z 596.291,A -85,B 0,C 180,E1 34247.431,E2 34247.431} C_VEL
LIN {X 0,Y 736.081,Z 596.285,A -85,B 0,C 180,E1 34244.502,E2 34244.502} C_VEL
LIN {X 0,Y 736.086,Z 596.289,A -85,B 0,C 180,E1 34241.625,E2 34241.625} C_VEL
LIN {X 0,Y 736.081,Z 596.286,A -85,B 0,C 180,E1 34238.765,E2 34238.765} C_VEL
LIN {X 0,Y 736.097,Z 596.287,A -85,B 0,C 180,E1 34235.835,E2 34235.835} C_VEL
LIN {X 0,Y 736.098,Z 596.285,A -85,B 0,C 180,E1 34232.727,E2 34232.727} C_VEL
LIN {X 0,Y 736.094,Z 596.29,A -85,B 0,C 180,E1 34229.723,E2 34229.723} C_VEL
LIN {X 0,Y 736.093,Z 596.357,A -85,B 0,C 180,E1 34227.386,E2 34227.386} C_VEL
LIN {X 0,Y 737.561,Z 601.435,A -85,B 0,C 180,E1 34226.932,E2 34226.932} C_VEL
LIN {X 0,Y 738.933,Z 607.122,A -85,B 0,C 180,E1 34226.808,E2 34226.808} C_VEL
LIN {X 0,Y 738.43,Z 864.226,A -85,B 0,C 180,E1 34224.044,E2 34224.044} C_VEL
LIN {X 0,Y 738.249,Z 946.976,A -85,B 0,C 180,E1 34223.145,E2 34223.145} C_VEL
LIN {X 0,Y 738.107,Z 971.005,A -85,B 0,C 180,E1 34222.74,E2 34222.74} C_VEL
LIN {X 0,Y 737.962,Z 992.64,A -85,B 0,C 180,E1 34222.241,E2 34222.241} C_VEL
LIN {X 0,Y 737.732,Z 1014.977,A -85,B 0,C 180,E1 34221.575,E2 34221.575} C_VEL
LIN {X 0,Y 737.57,Z 1036.263,A -85,B 0,C 180,E1 34220.805,E2 34220.805} C_VEL
LIN {X 0,Y 737.314,Z 1057.838,A -85,B 0,C 180,E1 34219.859,E2 34219.859} C_VEL
LIN {X 0,Y 737.074,Z 1078.545,A -85,B 0,C 180,E1 34218.795,E2 34218.795} C_VEL
LIN {X 0,Y 736.87,Z 1098.217,A -85,B 0,C 180,E1 34217.614,E2 34217.614} C_VEL
LIN {X 0,Y 736.639,Z 1116.823,A -85,B 0,C 180,E1 34216.319,E2 34216.319} C_VEL
LIN {X 0,Y 736.465,Z 1133.99,A -85,B 0,C 180,E1 34214.949,E2 34214.949} C_VEL
LIN {X 0,Y 736.316,Z 1149.696,A -85,B 0,C 180,E1 34213.507,E2 34213.507} C_VEL
LIN {X 0,Y 736.173,Z 1164.713,A -85,B 0,C 180,E1 34211.915,E2 34211.915} C_VEL
LIN {X 0,Y 736.076,Z 1177.649,A -85,B 0,C 180,E1 34210.33,E2 34210.33} C_VEL
LIN {X 0,Y 736.013,Z 1188.61,A -85,B 0,C 180,E1 34208.752,E2 34208.752} C_VEL
LIN {X 0,Y 735.972,Z 1198.842,A -85,B 0,C 180,E1 34207.023,E2 34207.023} C_VEL
LIN {X 0,Y 735.934,Z 1207.18,A -85,B 0,C 180,E1 34205.301,E2 34205.301} C_VEL
LIN {X 0,Y 735.915,Z 1214.077,A -85,B 0,C 180,E1 34203.505,E2 34203.505} C_VEL
LIN {X 0,Y 735.909,Z 1218.651,A -85,B 0,C 180,E1 34201.947,E2 34201.947} C_VEL
LIN {X 0,Y 735.915,Z 1222.506,A -85,B 0,C 180,E1 34200.078,E2 34200.078} C_VEL
LIN {X 0,Y 735.914,Z 1224.526,A -85,B 0,C 180,E1 34198.287,E2 34198.287} C_VEL
LIN {X 0,Y 735.913,Z 1224.871,A -85,B 0,C 180,E1 34196.495,E2 34196.495} C_VEL
LIN {X 0,Y 735.912,Z 1223.789,A -85,B 0,C 180,E1 34194.777,E2 34194.777} C_VEL
LIN {X 0,Y 735.909,Z 1220.956,A -85,B 0,C 180,E1 34192.976,E2 34192.976} C_VEL
LIN {X 0,Y 735.918,Z 1216.541,A -85,B 0,C 180,E1 34191.168,E2 34191.168} C_VEL
LIN {X 0,Y 735.914,Z 1210.538,A -85,B 0,C 180,E1 34189.431,E2 34189.431} C_VEL
LIN {X 0,Y 735.956,Z 1202.948,A -85,B 0,C 180,E1 34187.684,E2 34187.684} C_VEL
LIN {X 0,Y 735.987,Z 1193.852,A -85,B 0,C 180,E1 34186.006,E2 34186.006} C_VEL
LIN {X 0,Y 736.045,Z 1182.393,A -85,B 0,C 180,E1 34184.235,E2 34184.235} C_VEL
LIN {X 0,Y 736.136,Z 1170.661,A -85,B 0,C 180,E1 34182.694,E2 34182.694} C_VEL
LIN {X 0,Y 736.241,Z 1156.933,A -85,B 0,C 180,E1 34181.142,E2 34181.142} C_VEL
LIN {X 0,Y 736.403,Z 1141.913,A -85,B 0,C 180,E1 34179.659,E2 34179.659} C_VEL
LIN {X 0,Y 736.551,Z 1124.889,A -85,B 0,C 180,E1 34178.211,E2 34178.211} C_VEL
LIN {X 0,Y 736.754,Z 1106.687,A -85,B 0,C 180,E1 34176.865,E2 34176.865} C_VEL
LIN {X 0,Y 736.993,Z 1087.724,A -85,B 0,C 180,E1 34175.642,E2 34175.642} C_VEL
LIN {X 0,Y 737.2,Z 1066.838,A -85,B 0,C 180,E1 34174.492,E2 34174.492} C_VEL
LIN {X 0,Y 737.454,Z 1045.516,A -85,B 0,C 180,E1 34173.493,E2 34173.493} C_VEL
LIN {X 0,Y 737.667,Z 1024.081,A -85,B 0,C 180,E1 34172.645,E2 34172.645} C_VEL
LIN {X 0,Y 737.871,Z 1001.856,A -85,B 0,C 180,E1 34171.928,E2 34171.928} C_VEL
LIN {X 0,Y 738.035,Z 979.867,A -85,B 0,C 180,E1 34171.358,E2 34171.358} C_VEL
LIN {X 0,Y 738.196,Z 957.656,A -85,B 0,C 180,E1 34170.926,E2 34170.926} C_VEL
LIN {X 0,Y 738.304,Z 932.82,A -85,B 0,C 180,E1 34170.593,E2 34170.593} C_VEL
LIN {X 0,Y 738.799,Z 672.092,A -85,B 0,C 180,E1 34167.807,E2 34167.807} C_VEL
LIN {X 0,Y 738.726,Z 605.504,A -85,B 0,C 180,E1 34167.075,E2 34167.075} C_VEL
LIN {X 0,Y 737.327,Z 600.688,A -85,B 0,C 180,E1 34166.937,E2 34166.937} C_VEL
LIN {X 0,Y 736.081,Z 596.296,A -85,B 0,C 180,E1 34166.518,E2 34166.518} C_VEL
LIN {X 0,Y 736.094,Z 596.295,A -85,B 0,C 180,E1 34163.586,E2 34163.586} C_VEL
LIN {X 0,Y 736.094,Z 596.292,A -85,B 0,C 180,E1 34160.728,E2 34160.728} C_VEL
LIN {X 0,Y 736.091,Z 596.292,A -85,B 0,C 180,E1 34157.747,E2 34157.747} C_VEL
LIN {X 0,Y 736.104,Z 596.392,A -85,B 0,C 180,E1 34157.292,E2 34157.292} C_VEL
LIN {X 0,Y 736.552,Z 598.944,A -85,B 0,C 180,E1 34157.145,E2 34157.145} C_VEL
LIN {X 0,Y 736.091,Z 617.771,A -85,B 0,C 180,E1 34156.331,E2 34156.331} C_VEL
LIN {X 0,Y 735.922,Z 694.539,A -85,B 0,C 180,E1 34153.403,E2 34153.403} C_VEL
LIN {X 0,Y 735.915,Z 742.598,A -85,B 0,C 180,E1 34151.429,E2 34151.429} C_VEL
LIN {X 0,Y 736.671,Z 770.098,A -85,B 0,C 180,E1 34150.227,E2 34150.227} C_VEL
LIN {X 0,Y 738.862,Z 786.185,A -85,B 0,C 180,E1 34149.498,E2 34149.498} C_VEL
LIN {X 0,Y 741.013,Z 793.635,A -85,B 0,C 180,E1 34149.062,E2 34149.062} C_VEL
LIN {X 0,Y 743.475,Z 799.053,A -85,B 0,C 180,E1 34148.611,E2 34148.611} C_VEL
LIN {X 0,Y 746.111,Z 802.669,A -85,B 0,C 180,E1 34148.125,E2 34148.125} C_VEL
LIN {X 0,Y 748.17,Z 804.13,A -85,B 0,C 180,E1 34147.704,E2 34147.704} C_VEL
LIN {X 0,Y 749.938,Z 804.114,A -85,B 0,C 180,E1 34147.252,E2 34147.252} C_VEL
LIN {X 0,Y 751,Z 802.545,A -85,B 0,C 180,E1 34146.809,E2 34146.809} C_VEL
LIN {X 0,Y 751.147,Z 799.427,A -85,B 0,C 180,E1 34146.396,E2 34146.396} C_VEL
LIN {X 0,Y 750.317,Z 795.129,A -85,B 0,C 180,E1 34146.064,E2 34146.064} C_VEL
LIN {X 0,Y 748.54,Z 789.365,A -85,B 0,C 180,E1 34145.815,E2 34145.815} C_VEL
LIN {X 0,Y 746.698,Z 781.117,A -85,B 0,C 180,E1 34145.618,E2 34145.618} C_VEL
LIN {X 0,Y 745.78,Z 771.123,A -85,B 0,C 180,E1 34145.52,E2 34145.52} C_VEL
LIN {X 0,Y 745.589,Z 608.256,A -85,B 0,C 180,E1 34145.499,E2 34145.499} C_VEL
LIN {X 0,Y 742.41,Z 604.975,A -85,B 0,C 180,E1 34145.154,E2 34145.154} C_VEL
LIN {X 0,Y 741.117,Z 602.937,A -85,B 0,C 180,E1 34145.012,E2 34145.012} C_VEL
LIN {X 0,Y 739.256,Z 603.033,A -85,B 0,C 180,E1 34144.805,E2 34144.805} C_VEL
LIN {X 0,Y 738.051,Z 602.072,A -85,B 0,C 180,E1 34144.669,E2 34144.669} C_VEL
LIN {X 0,Y 738.43,Z 604.891,A -85,B 0,C 180,E1 34144.448,E2 34144.448} C_VEL
LIN {X 0,Y 738.086,Z 644.338,A -85,B 0,C 180,E1 34141.705,E2 34141.705} C_VEL
LIN {X 0,Y 737.93,Z 670.103,A -85,B 0,C 180,E1 34139.975,E2 34139.975} C_VEL
LIN {X 0,Y 738.952,Z 675.582,A -85,B 0,C 180,E1 34139.869,E2 34139.869} C_VEL
LIN {X 0,Y 738.395,Z 950.927,A -85,B 0,C 180,E1 34136.911,E2 34136.911} C_VEL
LIN {X 0,Y 738.243,Z 1018.689,A -85,B 0,C 180,E1 34136.171,E2 34136.171} C_VEL
LIN {X 0,Y 738.105,Z 1042.141,A -85,B 0,C 180,E1 34135.761,E2 34135.761} C_VEL
LIN {X 0,Y 737.942,Z 1064.217,A -85,B 0,C 180,E1 34135.245,E2 34135.245} C_VEL
LIN {X 0,Y 737.747,Z 1086.404,A -85,B 0,C 180,E1 34134.573,E2 34134.573} C_VEL
LIN {X 0,Y 737.535,Z 1108.026,A -85,B 0,C 180,E1 34133.778,E2 34133.778} C_VEL
LIN {X 0,Y 737.309,Z 1128.7,A -85,B 0,C 180,E1 34132.864,E2 34132.864} C_VEL
LIN {X 0,Y 737.041,Z 1150.311,A -85,B 0,C 180,E1 34131.739,E2 34131.739} C_VEL
LIN {X 0,Y 736.852,Z 1169.801,A -85,B 0,C 180,E1 34130.558,E2 34130.558} C_VEL
LIN {X 0,Y 736.634,Z 1188.212,A -85,B 0,C 180,E1 34129.26,E2 34129.26} C_VEL
LIN {X 0,Y 736.433,Z 1206.324,A -85,B 0,C 180,E1 34127.789,E2 34127.789} C_VEL
LIN {X 0,Y 736.299,Z 1221.989,A -85,B 0,C 180,E1 34126.327,E2 34126.327} C_VEL
LIN {X 0,Y 736.173,Z 1236.15,A -85,B 0,C 180,E1 34124.795,E2 34124.795} C_VEL
LIN {X 0,Y 736.069,Z 1249.671,A -85,B 0,C 180,E1 34123.096,E2 34123.096} C_VEL
LIN {X 0,Y 736.02,Z 1260.425,A -85,B 0,C 180,E1 34121.52,E2 34121.52} C_VEL
LIN {X 0,Y 735.953,Z 1270.336,A -85,B 0,C 180,E1 34119.779,E2 34119.779} C_VEL
LIN {X 0,Y 735.932,Z 1278.51,A -85,B 0,C 180,E1 34118.046,E2 34118.046} C_VEL
LIN {X 0,Y 735.92,Z 1284.822,A -85,B 0,C 180,E1 34116.319,E2 34116.319} C_VEL
LIN {X 0,Y 735.895,Z 1289.667,A -85,B 0,C 180,E1 34114.599,E2 34114.599} C_VEL
LIN {X 0,Y 735.898,Z 1292.963,A -85,B 0,C 180,E1 34112.805,E2 34112.805} C_VEL
LIN {X 0,Y 735.914,Z 1294.714,A -85,B 0,C 180,E1 34111.013,E2 34111.013} C_VEL
LIN {X 0,Y 735.892,Z 1294.829,A -85,B 0,C 180,E1 34109.378,E2 34109.378} C_VEL
LIN {X 0,Y 735.895,Z 1293.526,A -85,B 0,C 180,E1 34107.587,E2 34107.587} C_VEL
LIN {X 0,Y 735.913,Z 1290.479,A -85,B 0,C 180,E1 34105.786,E2 34105.786} C_VEL
LIN {X 0,Y 735.919,Z 1285.585,A -85,B 0,C 180,E1 34103.918,E2 34103.918} C_VEL
LIN {X 0,Y 735.914,Z 1279.745,A -85,B 0,C 180,E1 34102.271,E2 34102.271} C_VEL
LIN {X 0,Y 735.957,Z 1271.569,A -85,B 0,C 180,E1 34100.46,E2 34100.46} C_VEL
LIN {X 0,Y 736.009,Z 1261.929,A -85,B 0,C 180,E1 34098.72,E2 34098.72} C_VEL
LIN {X 0,Y 736.061,Z 1250.714,A -85,B 0,C 180,E1 34097.049,E2 34097.049} C_VEL
LIN {X 0,Y 736.158,Z 1238.288,A -85,B 0,C 180,E1 34095.448,E2 34095.448} C_VEL
LIN {X 0,Y 736.271,Z 1223.578,A -85,B 0,C 180,E1 34093.837,E2 34093.837} C_VEL
LIN {X 0,Y 736.415,Z 1208.202,A -85,B 0,C 180,E1 34092.376,E2 34092.376} C_VEL
LIN {X 0,Y 736.61,Z 1191.534,A -85,B 0,C 180,E1 34090.989,E2 34090.989} C_VEL
LIN {X 0,Y 736.817,Z 1172.02,A -85,B 0,C 180,E1 34089.59,E2 34089.59} C_VEL
LIN {X 0,Y 737.029,Z 1152.536,A -85,B 0,C 180,E1 34088.389,E2 34088.389} C_VEL
LIN {X 0,Y 737.284,Z 1132.274,A -85,B 0,C 180,E1 34087.306,E2 34087.306} C_VEL
LIN {X 0,Y 737.475,Z 1111.864,A -85,B 0,C 180,E1 34086.383,E2 34086.383} C_VEL
LIN {X 0,Y 737.726,Z 1089.835,A -85,B 0,C 180,E1 34085.541,E2 34085.541} C_VEL
LIN {X 0,Y 737.882,Z 1068.542,A -85,B 0,C 180,E1 34084.877,E2 34084.877} C_VEL
LIN {X 0,Y 738.101,Z 1044.824,A -85,B 0,C 180,E1 34084.294,E2 34084.294} C_VEL
LIN {X 0,Y 738.201,Z 1022.197,A -85,B 0,C 180,E1 34083.882,E2 34083.882} C_VEL
LIN {X 0,Y 738.308,Z 990.543,A -85,B 0,C 180,E1 34083.508,E2 34083.508} C_VEL
LIN {X 0,Y 738.84,Z 731.406,A -85,B 0,C 180,E1 34080.737,E2 34080.737} C_VEL
LIN {X 0,Y 738.745,Z 673.594,A -85,B 0,C 180,E1 34080.1,E2 34080.1} C_VEL
LIN {X 0,Y 737.853,Z 669.306,A -85,B 0,C 180,E1 34079.99,E2 34079.99} C_VEL
LIN {X 0,Y 738.243,Z 627.195,A -85,B 0,C 180,E1 34077.113,E2 34077.113} C_VEL
LIN {X 0,Y 738.371,Z 603.104,A -85,B 0,C 180,E1 34075.421,E2 34075.421} C_VEL
LIN {X 0,Y 738.101,Z 602.133,A -85,B 0,C 180,E1 34075.324,E2 34075.324} C_VEL
LIN {X 0,Y 739.812,Z 603.167,A -85,B 0,C 180,E1 34075.133,E2 34075.133} C_VEL
LIN {X 0,Y 741.316,Z 603.094,A -85,B 0,C 180,E1 34074.966,E2 34074.966} C_VEL
LIN {X 0,Y 743.835,Z 606.74,A -85,B 0,C 180,E1 34074.69,E2 34074.69} C_VEL
LIN {X 0,Y 745.694,Z 608.328,A -85,B 0,C 180,E1 34074.489,E2 34074.489} C_VEL
LIN {X 0,Y 745.846,Z 772.595,A -85,B 0,C 180,E1 34074.473,E2 34074.473} C_VEL
LIN {X 0,Y 746.9,Z 782.362,A -85,B 0,C 180,E1 34074.36,E2 34074.36} C_VEL
LIN {X 0,Y 748.927,Z 790.61,A -85,B 0,C 180,E1 34074.144,E2 34074.144} C_VEL
LIN {X 0,Y 750.505,Z 795.882,A -85,B 0,C 180,E1 34073.89,E2 34073.89} C_VEL
LIN {X 0,Y 751.196,Z 800.053,A -85,B 0,C 180,E1 34073.538,E2 34073.538} C_VEL
LIN {X 0,Y 750.941,Z 802.744,A -85,B 0,C 180,E1 34073.154,E2 34073.154} C_VEL
LIN {X 0,Y 749.938,Z 804.114,A -85,B 0,C 180,E1 34072.748,E2 34072.748} C_VEL
LIN {X 0,Y 748.169,Z 804.131,A -85,B 0,C 180,E1 34072.296,E2 34072.296} C_VEL
LIN {X 0,Y 745.884,Z 802.444,A -85,B 0,C 180,E1 34071.832,E2 34071.832} C_VEL
LIN {X 0,Y 743.472,Z 799.045,A -85,B 0,C 180,E1 34071.388,E2 34071.388} C_VEL
LIN {X 0,Y 740.392,Z 791.301,A -85,B 0,C 180,E1 34070.699,E2 34070.699} C_VEL
LIN {X 0,Y 738.78,Z 780.714,A -85,B 0,C 180,E1 34069.88,E2 34069.88} C_VEL
LIN {X 0,Y 738.883,Z 728.426,A -85,B 0,C 180,E1 34066.145,E2 34066.145} C_VEL
LIN {X 0,Y 739.298,Z 691.63,A -85,B 0,C 180,E1 34063.427,E2 34063.427} C_VEL
LIN {X 0,Y 739.707,Z 655.865,A -85,B 0,C 180,E1 34060.686,E2 34060.686} C_VEL
LIN {X 0,Y 740.086,Z 620.939,A -85,B 0,C 180,E1 34057.91,E2 34057.91} C_VEL
LIN {X 0,Y 740.122,Z 606.307,A -85,B 0,C 180,E1 34056.713,E2 34056.713} C_VEL
LIN {X 0,Y 737.07,Z 599.24,A -85,B 0,C 180,E1 34055.877,E2 34055.877} C_VEL
LIN {X 0,Y 736.094,Z 596.283,A -85,B 0,C 180,E1 34055.522,E2 34055.522} C_VEL
LIN {X 0,Y 736.098,Z 596.291,A -85,B 0,C 180,E1 34052.542,E2 34052.542} C_VEL
LIN {X 0,Y 736.092,Z 596.29,A -85,B 0,C 180,E1 34049.544,E2 34049.544} C_VEL
LIN {X 0,Y 736.1,Z 596.288,A -85,B 0,C 180,E1 34046.475,E2 34046.475} C_VEL
LIN {X 0,Y 736.097,Z 596.287,A -85,B 0,C 180,E1 34043.453,E2 34043.453} C_VEL
LIN {X 0,Y 736.093,Z 596.287,A -85,B 0,C 180,E1 34040.406,E2 34040.406} C_VEL
LIN {X 0,Y 736.078,Z 596.289,A -85,B 0,C 180,E1 34037.47,E2 34037.47} C_VEL
LIN {X 0,Y 736.092,Z 596.292,A -85,B 0,C 180,E1 34034.635,E2 34034.635} C_VEL
LIN {X 0,Y 736.1,Z 596.294,A -85,B 0,C 180,E1 34031.665,E2 34031.665} C_VEL
LIN {X 0,Y 736.093,Z 596.29,A -85,B 0,C 180,E1 34028.751,E2 34028.751} C_VEL
LIN {X 0,Y 736.096,Z 596.286,A -85,B 0,C 180,E1 34025.769,E2 34025.769} C_VEL
LIN {X 0,Y 736.09,Z 596.287,A -85,B 0,C 180,E1 34022.725,E2 34022.725} C_VEL
LIN {X 0,Y 736.079,Z 596.288,A -85,B 0,C 180,E1 34019.766,E2 34019.766} C_VEL
LIN {X 0,Y 736.073,Z 596.291,A -85,B 0,C 180,E1 34016.885,E2 34016.885} C_VEL
LIN {X 0,Y 736.094,Z 596.293,A -85,B 0,C 180,E1 34014.074,E2 34014.074} C_VEL
LIN {X 0,Y 736.098,Z 596.291,A -85,B 0,C 180,E1 34011.17,E2 34011.17} C_VEL
LIN {X 0,Y 736.098,Z 596.289,A -85,B 0,C 180,E1 34009.084,E2 34009.084} C_VEL
LIN {X 0,Y 735.093,Z 596.413,A -85,B 0,C 180,E1 34008.485,E2 34008.485} C_VEL
LIN {X 0,Y 728.671,Z 597.213,A -85,B 0,C 180,E1 34006.806,E2 34006.806} C_VEL
LIN {X 0,Y 728.153,Z 597.28,A -85,B 0,C 180,E1 34006.369,E2 34006.369} C_VEL
LIN {X 0,Y 728.136,Z 597.279,A -85,B 0,C 180,E1 34003.485,E2 34003.485} C_VEL
LIN {X 0,Y 728.151,Z 597.276,A -85,B 0,C 180,E1 34000.591,E2 34000.591} C_VEL
LIN {X 0,Y 728.154,Z 597.276,A -85,B 0,C 180,E1 33997.558,E2 33997.558} C_VEL
LIN {X 0,Y 728.157,Z 597.276,A -85,B 0,C 180,E1 33994.545,E2 33994.545} C_VEL
LIN {X 0,Y 728.156,Z 597.277,A -85,B 0,C 180,E1 33991.454,E2 33991.454} C_VEL
LIN {X 0,Y 728.16,Z 597.278,A -85,B 0,C 180,E1 33988.454,E2 33988.454} C_VEL
LIN {X 0,Y 728.15,Z 597.282,A -85,B 0,C 180,E1 33985.476,E2 33985.476} C_VEL
LIN {X 0,Y 728.138,Z 597.282,A -85,B 0,C 180,E1 33982.63,E2 33982.63} C_VEL
LIN {X 0,Y 728.153,Z 597.276,A -85,B 0,C 180,E1 33979.77,E2 33979.77} C_VEL
LIN {X 0,Y 728.153,Z 597.271,A -85,B 0,C 180,E1 33976.747,E2 33976.747} C_VEL
LIN {X 0,Y 728.158,Z 597.275,A -85,B 0,C 180,E1 33973.684,E2 33973.684} C_VEL
LIN {X 0,Y 728.162,Z 597.275,A -85,B 0,C 180,E1 33970.592,E2 33970.592} C_VEL
LIN {X 0,Y 728.159,Z 597.274,A -85,B 0,C 180,E1 33967.466,E2 33967.466} C_VEL
LIN {X 0,Y 728.158,Z 597.275,A -85,B 0,C 180,E1 33964.357,E2 33964.357} C_VEL
LIN {X 0,Y 728.163,Z 597.279,A -85,B 0,C 180,E1 33961.267,E2 33961.267} C_VEL
LIN {X 0,Y 728.185,Z 597.458,A -85,B 0,C 180,E1 33959.002,E2 33959.002} C_VEL
LIN {X 0,Y 729.994,Z 604.227,A -85,B 0,C 180,E1 33958.511,E2 33958.511} C_VEL
LIN {X 0,Y 730.027,Z 640.636,A -85,B 0,C 180,E1 33956.216,E2 33956.216} C_VEL
LIN {X 0,Y 729.678,Z 684.164,A -85,B 0,C 180,E1 33953.414,E2 33953.414} C_VEL
LIN {X 0,Y 729.287,Z 729.572,A -85,B 0,C 180,E1 33950.539,E2 33950.539} C_VEL
LIN {X 0,Y 728.949,Z 776.127,A -85,B 0,C 180,E1 33947.645,E2 33947.645} C_VEL
LIN {X 0,Y 728.652,Z 823.513,A -85,B 0,C 180,E1 33944.746,E2 33944.746} C_VEL
LIN {X 0,Y 728.656,Z 831.032,A -85,B 0,C 180,E1 33944.309,E2 33944.309} C_VEL
LIN {X 0,Y 728.981,Z 840.58,A -85,B 0,C 180,E1 33944.206,E2 33944.206} C_VEL
LIN {X 0,Y 728.745,Z 1001.113,A -85,B 0,C 180,E1 33942.59,E2 33942.59} C_VEL
LIN {X 0,Y 728.678,Z 1018.938,A -85,B 0,C 180,E1 33942.254,E2 33942.254} C_VEL
LIN {X 0,Y 728.578,Z 1035.424,A -85,B 0,C 180,E1 33941.798,E2 33941.798} C_VEL
LIN {X 0,Y 728.472,Z 1051.617,A -85,B 0,C 180,E1 33941.198,E2 33941.198} C_VEL
LIN {X 0,Y 728.364,Z 1066.811,A -85,B 0,C 180,E1 33940.479,E2 33940.479} C_VEL
LIN {X 0,Y 728.239,Z 1081.571,A -85,B 0,C 180,E1 33939.602,E2 33939.602} C_VEL
LIN {X 0,Y 728.142,Z 1095.157,A -85,B 0,C 180,E1 33938.607,E2 33938.607} C_VEL
LIN {X 0,Y 728.062,Z 1106.666,A -85,B 0,C 180,E1 33937.575,E2 33937.575} C_VEL
LIN {X 0,Y 727.997,Z 1117.38,A -85,B 0,C 180,E1 33936.386,E2 33936.386} C_VEL
LIN {X 0,Y 727.954,Z 1126.473,A -85,B 0,C 180,E1 33935.121,E2 33935.121} C_VEL
LIN {X 0,Y 727.932,Z 1133.521,A -85,B 0,C 180,E1 33933.858,E2 33933.858} C_VEL
LIN {X 0,Y 727.92,Z 1139.015,A -85,B 0,C 180,E1 33932.518,E2 33932.518} C_VEL
LIN {X 0,Y 727.913,Z 1142.662,A -85,B 0,C 180,E1 33931.18,E2 33931.18} C_VEL
LIN {X 0,Y 727.914,Z 1144.665,A -85,B 0,C 180,E1 33929.763,E2 33929.763} C_VEL
LIN {X 0,Y 727.915,Z 1144.857,A -85,B 0,C 180,E1 33928.425,E2 33928.425} C_VEL
LIN {X 0,Y 727.916,Z 1143.37,A -85,B 0,C 180,E1 33927.086,E2 33927.086} C_VEL
LIN {X 0,Y 727.919,Z 1140.143,A -85,B 0,C 180,E1 33925.745,E2 33925.745} C_VEL
LIN {X 0,Y 727.926,Z 1135.116,A -85,B 0,C 180,E1 33924.402,E2 33924.402} C_VEL
LIN {X 0,Y 727.945,Z 1128.589,A -85,B 0,C 180,E1 33923.136,E2 33923.136} C_VEL
LIN {X 0,Y 727.985,Z 1120.092,A -85,B 0,C 180,E1 33921.866,E2 33921.866} C_VEL
LIN {X 0,Y 728.041,Z 1109.942,A -85,B 0,C 180,E1 33920.673,E2 33920.673} C_VEL
LIN {X 0,Y 728.116,Z 1098.17,A -85,B 0,C 180,E1 33919.555,E2 33919.555} C_VEL
LIN {X 0,Y 728.218,Z 1085.254,A -85,B 0,C 180,E1 33918.555,E2 33918.555} C_VEL
LIN {X 0,Y 728.325,Z 1071.187,A -85,B 0,C 180,E1 33917.673,E2 33917.673} C_VEL
LIN {X 0,Y 728.43,Z 1056.104,A -85,B 0,C 180,E1 33916.909,E2 33916.909} C_VEL
LIN {X 0,Y 728.542,Z 1039.966,A -85,B 0,C 180,E1 33916.264,E2 33916.264} C_VEL
LIN {X 0,Y 728.655,Z 1023.02,A -85,B 0,C 180,E1 33915.755,E2 33915.755} C_VEL
LIN {X 0,Y 728.738,Z 1005.006,A -85,B 0,C 180,E1 33915.381,E2 33915.381} C_VEL
LIN {X 0,Y 728.785,Z 982.538,A -85,B 0,C 180,E1 33915.115,E2 33915.115} C_VEL
LIN {X 0,Y 728.757,Z 831.804,A -85,B 0,C 180,E1 33913.611,E2 33913.611} C_VEL
LIN {X 0,Y 728.613,Z 830.325,A -85,B 0,C 180,E1 33913.578,E2 33913.578} C_VEL
LIN {X 0,Y 728.914,Z 782.423,A -85,B 0,C 180,E1 33910.653,E2 33910.653} C_VEL
LIN {X 0,Y 729.271,Z 733.12,A -85,B 0,C 180,E1 33907.594,E2 33907.594} C_VEL
LIN {X 0,Y 729.626,Z 688.192,A -85,B 0,C 180,E1 33904.753,E2 33904.753} C_VEL
LIN {X 0,Y 730.022,Z 645.128,A -85,B 0,C 180,E1 33901.978,E2 33901.978} C_VEL
LIN {X 0,Y 729.997,Z 603.906,A -85,B 0,C 180,E1 33899.378,E2 33899.378} C_VEL
LIN {X 0,Y 728.164,Z 597.282,A -85,B 0,C 180,E1 33898.868,E2 33898.868} C_VEL
LIN {X 0,Y 728.148,Z 597.271,A -85,B 0,C 180,E1 33895.83,E2 33895.83} C_VEL
LIN {X 0,Y 728.157,Z 597.279,A -85,B 0,C 180,E1 33892.828,E2 33892.828} C_VEL
LIN {X 0,Y 728.134,Z 597.271,A -85,B 0,C 180,E1 33889.905,E2 33889.905} C_VEL
LIN {X 0,Y 728.151,Z 597.281,A -85,B 0,C 180,E1 33887.047,E2 33887.047} C_VEL
LIN {X 0,Y 728.153,Z 597.272,A -85,B 0,C 180,E1 33884.095,E2 33884.095} C_VEL
LIN {X 0,Y 728.156,Z 597.278,A -85,B 0,C 180,E1 33881.025,E2 33881.025} C_VEL
LIN {X 0,Y 728.156,Z 597.273,A -85,B 0,C 180,E1 33878.066,E2 33878.066} C_VEL
LIN {X 0,Y 728.148,Z 597.279,A -85,B 0,C 180,E1 33875.03,E2 33875.03} C_VEL
LIN {X 0,Y 728.136,Z 597.278,A -85,B 0,C 180,E1 33872.196,E2 33872.196} C_VEL
LIN {X 0,Y 728.139,Z 597.279,A -85,B 0,C 180,E1 33869.309,E2 33869.309} C_VEL
LIN {X 0,Y 728.173,Z 597.414,A -85,B 0,C 180,E1 33867.664,E2 33867.664} C_VEL
LIN {X 0,Y 729.325,Z 601.448,A -85,B 0,C 180,E1 33867.306,E2 33867.306} C_VEL
LIN {X 0,Y 731.715,Z 606.87,A -85,B 0,C 180,E1 33867.136,E2 33867.136} C_VEL
LIN {X 0,Y 731.975,Z 612.687,A -85,B 0,C 180,E1 33867.059,E2 33867.059} C_VEL
LIN {X 0,Y 731.29,Z 869.596,A -85,B 0,C 180,E1 33864.272,E2 33864.272} C_VEL
LIN {X 0,Y 731.059,Z 946.954,A -85,B 0,C 180,E1 33863.422,E2 33863.422} C_VEL
LIN {X 0,Y 730.871,Z 971.113,A -85,B 0,C 180,E1 33863.012,E2 33863.012} C_VEL
LIN {X 0,Y 730.66,Z 993.449,A -85,B 0,C 180,E1 33862.488,E2 33862.488} C_VEL
LIN {X 0,Y 730.371,Z 1015.451,A -85,B 0,C 180,E1 33861.824,E2 33861.824} C_VEL
LIN {X 0,Y 730.119,Z 1037.819,A -85,B 0,C 180,E1 33860.999,E2 33860.999} C_VEL
LIN {X 0,Y 729.792,Z 1059.474,A -85,B 0,C 180,E1 33860.031,E2 33860.031} C_VEL
LIN {X 0,Y 729.45,Z 1080.529,A -85,B 0,C 180,E1 33858.92,E2 33858.92} C_VEL
LIN {X 0,Y 729.173,Z 1100.635,A -85,B 0,C 180,E1 33857.682,E2 33857.682} C_VEL
LIN {X 0,Y 728.882,Z 1118.929,A -85,B 0,C 180,E1 33856.374,E2 33856.374} C_VEL
LIN {X 0,Y 728.627,Z 1136.221,A -85,B 0,C 180,E1 33854.951,E2 33854.951} C_VEL
LIN {X 0,Y 728.436,Z 1152.46,A -85,B 0,C 180,E1 33853.414,E2 33853.414} C_VEL
LIN {X 0,Y 728.264,Z 1166.415,A -85,B 0,C 180,E1 33851.885,E2 33851.885} C_VEL
LIN {X 0,Y 728.121,Z 1179.628,A -85,B 0,C 180,E1 33850.204,E2 33850.204} C_VEL
LIN {X 0,Y 728.038,Z 1190.887,A -85,B 0,C 180,E1 33848.53,E2 33848.53} C_VEL
LIN {X 0,Y 727.981,Z 1200.765,A -85,B 0,C 180,E1 33846.758,E2 33846.758} C_VEL
LIN {X 0,Y 727.946,Z 1208.999,A -85,B 0,C 180,E1 33844.964,E2 33844.964} C_VEL
LIN {X 0,Y 727.92,Z 1215.196,A -85,B 0,C 180,E1 33843.229,E2 33843.229} C_VEL
LIN {X 0,Y 727.903,Z 1220.231,A -85,B 0,C 180,E1 33841.338,E2 33841.338} C_VEL
LIN {X 0,Y 727.907,Z 1223.228,A -85,B 0,C 180,E1 33839.606,E2 33839.606} C_VEL
LIN {X 0,Y 727.9,Z 1224.797,A -85,B 0,C 180,E1 33837.717,E2 33837.717} C_VEL
LIN {X 0,Y 727.913,Z 1224.725,A -85,B 0,C 180,E1 33835.983,E2 33835.983} C_VEL
LIN {X 0,Y 727.916,Z 1223.032,A -85,B 0,C 180,E1 33834.166,E2 33834.166} C_VEL
LIN {X 0,Y 727.915,Z 1219.757,A -85,B 0,C 180,E1 33832.343,E2 33832.343} C_VEL
LIN {X 0,Y 727.921,Z 1214.898,A -85,B 0,C 180,E1 33830.592,E2 33830.592} C_VEL
LIN {X 0,Y 727.94,Z 1208.86,A -85,B 0,C 180,E1 33828.913,E2 33828.913} C_VEL
LIN {X 0,Y 727.968,Z 1200.726,A -85,B 0,C 180,E1 33827.143,E2 33827.143} C_VEL
LIN {X 0,Y 728.031,Z 1190.761,A -85,B 0,C 180,E1 33825.362,E2 33825.362} C_VEL
LIN {X 0,Y 728.122,Z 1180.382,A -85,B 0,C 180,E1 33823.813,E2 33823.813} C_VEL
LIN {X 0,Y 728.26,Z 1167.683,A -85,B 0,C 180,E1 33822.171,E2 33822.171} C_VEL
LIN {X 0,Y 728.431,Z 1152.652,A -85,B 0,C 180,E1 33820.515,E2 33820.515} C_VEL
LIN {X 0,Y 728.617,Z 1136.801,A -85,B 0,C 180,E1 33819.012,E2 33819.012} C_VEL
LIN {X 0,Y 728.879,Z 1119.917,A -85,B 0,C 180,E1 33817.61,E2 33817.61} C_VEL
LIN {X 0,Y 729.177,Z 1100.617,A -85,B 0,C 180,E1 33816.225,E2 33816.225} C_VEL
LIN {X 0,Y 729.439,Z 1081.143,A -85,B 0,C 180,E1 33815.027,E2 33815.027} C_VEL
LIN {X 0,Y 729.774,Z 1061.212,A -85,B 0,C 180,E1 33813.962,E2 33813.962} C_VEL
LIN {X 0,Y 730.068,Z 1039.899,A -85,B 0,C 180,E1 33812.998,E2 33812.998} C_VEL
LIN {X 0,Y 730.351,Z 1017.911,A -85,B 0,C 180,E1 33812.17,E2 33812.17} C_VEL
LIN {X 0,Y 730.596,Z 997.55,A -85,B 0,C 180,E1 33811.535,E2 33811.535} C_VEL
LIN {X 0,Y 730.852,Z 974.384,A -85,B 0,C 180,E1 33810.965,E2 33810.965} C_VEL
LIN {X 0,Y 731.047,Z 949.65,A -85,B 0,C 180,E1 33810.523,E2 33810.523} C_VEL
LIN {X 0,Y 731.197,Z 905.611,A -85,B 0,C 180,E1 33810.024,E2 33810.024} C_VEL
LIN {X 0,Y 731.933,Z 634.541,A -85,B 0,C 180,E1 33807.091,E2 33807.091} C_VEL
LIN {X 0,Y 731.807,Z 607.278,A -85,B 0,C 180,E1 33806.783,E2 33806.783} C_VEL
LIN {X 0,Y 730.484,Z 603.889,A -85,B 0,C 180,E1 33806.685,E2 33806.685} C_VEL
LIN {X 0,Y 729.052,Z 600.71,A -85,B 0,C 180,E1 33806.563,E2 33806.563} C_VEL
LIN {X 0,Y 728.155,Z 597.28,A -85,B 0,C 180,E1 33806.211,E2 33806.211} C_VEL
LIN {X 0,Y 728.162,Z 597.279,A -85,B 0,C 180,E1 33803.124,E2 33803.124} C_VEL
LIN {X 0,Y 728.148,Z 597.283,A -85,B 0,C 180,E1 33800.112,E2 33800.112} C_VEL
LIN {X 0,Y 728.162,Z 597.443,A -85,B 0,C 180,E1 33797.563,E2 33797.563} C_VEL
LIN {X 0,Y 729.052,Z 600.758,A -85,B 0,C 180,E1 33797.318,E2 33797.318} C_VEL
LIN {X 0,Y 728.337,Z 616.559,A -85,B 0,C 180,E1 33796.544,E2 33796.544} C_VEL
LIN {X 0,Y 728.008,Z 649.534,A -85,B 0,C 180,E1 33795.204,E2 33795.204} C_VEL
LIN {X 0,Y 727.923,Z 708.603,A -85,B 0,C 180,E1 33792.866,E2 33792.866} C_VEL
LIN {X 0,Y 728.228,Z 761.997,A -85,B 0,C 180,E1 33790.598,E2 33790.598} C_VEL
LIN {X 0,Y 729.768,Z 780.371,A -85,B 0,C 180,E1 33789.767,E2 33789.767} C_VEL
LIN {X 0,Y 732.264,Z 792.583,A -85,B 0,C 180,E1 33789.214,E2 33789.214} C_VEL
LIN {X 0,Y 735.235,Z 800.487,A -85,B 0,C 180,E1 33788.807,E2 33788.807} C_VEL
LIN {X 0,Y 738.49,Z 806.037,A -85,B 0,C 180,E1 33788.376,E2 33788.376} C_VEL
LIN {X 0,Y 741.65,Z 809.399,A -85,B 0,C 180,E1 33787.936,E2 33787.936} C_VEL
LIN {X 0,Y 744.54,Z 810.963,A -85,B 0,C 180,E1 33787.468,E2 33787.468} C_VEL
LIN {X 0,Y 746.587,Z 810.886,A -85,B 0,C 180,E1 33787.04,E2 33787.04} C_VEL
LIN {X 0,Y 747.939,Z 809.435,A -85,B 0,C 180,E1 33786.602,E2 33786.602} C_VEL
LIN {X 0,Y 748.341,Z 806.554,A -85,B 0,C 180,E1 33786.177,E2 33786.177} C_VEL
LIN {X 0,Y 747.601,Z 802.336,A -85,B 0,C 180,E1 33785.802,E2 33785.802} C_VEL
LIN {X 0,Y 745.735,Z 796.989,A -85,B 0,C 180,E1 33785.515,E2 33785.515} C_VEL
LIN {X 0,Y 743.203,Z 788.437,A -85,B 0,C 180,E1 33785.24,E2 33785.24} C_VEL
LIN {X 0,Y 741.637,Z 778.542,A -85,B 0,C 180,E1 33785.069,E2 33785.069} C_VEL
LIN {X 0,Y 741.083,Z 767.615,A -85,B 0,C 180,E1 33785.008,E2 33785.008} C_VEL
LIN {X 0,Y 740.973,Z 613.063,A -85,B 0,C 180,E1 33784.996,E2 33784.996} C_VEL
LIN {X 0,Y 739.471,Z 611.276,A -85,B 0,C 180,E1 33784.829,E2 33784.829} C_VEL
LIN {X 0,Y 735.849,Z 616.555,A -85,B 0,C 180,E1 33784.422,E2 33784.422} C_VEL
LIN {X 0,Y 733.315,Z 618.656,A -85,B 0,C 180,E1 33784.132,E2 33784.132} C_VEL
LIN {X 0,Y 731.636,Z 618.664,A -85,B 0,C 180,E1 33783.937,E2 33783.937} C_VEL
LIN {X 0,Y 731.173,Z 618.281,A -85,B 0,C 180,E1 33783.879,E2 33783.879} C_VEL
LIN {X 0,Y 730.675,Z 659.411,A -85,B 0,C 180,E1 33781.017,E2 33781.017} C_VEL
LIN {X 0,Y 730.613,Z 670.092,A -85,B 0,C 180,E1 33780.307,E2 33780.307} C_VEL
LIN {X 0,Y 732.004,Z 677.087,A -85,B 0,C 180,E1 33780.165,E2 33780.165} C_VEL
LIN {X 0,Y 731.255,Z 951.691,A -85,B 0,C 180,E1 33777.187,E2 33777.187} C_VEL
LIN {X 0,Y 731.055,Z 1018.698,A -85,B 0,C 180,E1 33776.448,E2 33776.448} C_VEL
LIN {X 0,Y 730.865,Z 1042.464,A -85,B 0,C 180,E1 33776.029,E2 33776.029} C_VEL
LIN {X 0,Y 730.64,Z 1064.972,A -85,B 0,C 180,E1 33775.494,E2 33775.494} C_VEL
LIN {X 0,Y 730.383,Z 1087.004,A -85,B 0,C 180,E1 33774.818,E2 33774.818} C_VEL
LIN {X 0,Y 730.069,Z 1109.826,A -85,B 0,C 180,E1 33773.96,E2 33773.96} C_VEL
LIN {X 0,Y 729.776,Z 1131.366,A -85,B 0,C 180,E1 33772.986,E2 33772.986} C_VEL
LIN {X 0,Y 729.422,Z 1152.169,A -85,B 0,C 180,E1 33771.869,E2 33771.869} C_VEL
LIN {X 0,Y 729.145,Z 1171.994,A -85,B 0,C 180,E1 33770.637,E2 33770.637} C_VEL
LIN {X 0,Y 728.859,Z 1191.503,A -85,B 0,C 180,E1 33769.224,E2 33769.224} C_VEL
LIN {X 0,Y 728.6,Z 1208.181,A -85,B 0,C 180,E1 33767.821,E2 33767.821} C_VEL
LIN {X 0,Y 728.396,Z 1224.337,A -85,B 0,C 180,E1 33766.263,E2 33766.263} C_VEL
LIN {X 0,Y 728.241,Z 1238.93,A -85,B 0,C 180,E1 33764.634,E2 33764.634} C_VEL
LIN {X 0,Y 728.115,Z 1251.283,A -85,B 0,C 180,E1 33763.016,E2 33763.016} C_VEL
LIN {X 0,Y 728.036,Z 1262.547,A -85,B 0,C 180,E1 33761.299,E2 33761.299} C_VEL
LIN {X 0,Y 727.974,Z 1272.155,A -85,B 0,C 180,E1 33759.531,E2 33759.531} C_VEL
LIN {X 0,Y 727.92,Z 1280.034,A -85,B 0,C 180,E1 33757.737,E2 33757.737} C_VEL
LIN {X 0,Y 727.921,Z 1285.837,A -85,B 0,C 180,E1 33756.072,E2 33756.072} C_VEL
LIN {X 0,Y 727.914,Z 1290.653,A -85,B 0,C 180,E1 33754.176,E2 33754.176} C_VEL
LIN {X 0,Y 727.897,Z 1293.621,A -85,B 0,C 180,E1 33752.363,E2 33752.363} C_VEL
LIN {X 0,Y 727.893,Z 1294.829,A -85,B 0,C 180,E1 33750.631,E2 33750.631} C_VEL
LIN {X 0,Y 727.91,Z 1294.684,A -85,B 0,C 180,E1 33748.899,E2 33748.899} C_VEL
LIN {X 0,Y 727.909,Z 1292.76,A -85,B 0,C 180,E1 33747.019,E2 33747.019} C_VEL
LIN {X 0,Y 727.904,Z 1289.084,A -85,B 0,C 180,E1 33745.116,E2 33745.116} C_VEL
LIN {X 0,Y 727.907,Z 1284.316,A -85,B 0,C 180,E1 33743.454,E2 33743.454} C_VEL
LIN {X 0,Y 727.949,Z 1277.481,A -85,B 0,C 180,E1 33741.629,E2 33741.629} C_VEL
LIN {X 0,Y 727.987,Z 1269.132,A -85,B 0,C 180,E1 33739.876,E2 33739.876} C_VEL
LIN {X 0,Y 728.055,Z 1258.884,A -85,B 0,C 180,E1 33738.113,E2 33738.113} C_VEL
LIN {X 0,Y 728.157,Z 1247.542,A -85,B 0,C 180,E1 33736.462,E2 33736.462} C_VEL
LIN {X 0,Y 728.271,Z 1234.057,A -85,B 0,C 180,E1 33734.799,E2 33734.799} C_VEL
LIN {X 0,Y 728.464,Z 1219.555,A -85,B 0,C 180,E1 33733.248,E2 33733.248} C_VEL
LIN {X 0,Y 728.687,Z 1203.043,A -85,B 0,C 180,E1 33731.723,E2 33731.723} C_VEL
LIN {X 0,Y 728.912,Z 1185.761,A -85,B 0,C 180,E1 33730.342,E2 33730.342} C_VEL
LIN {X 0,Y 729.212,Z 1166.935,A -85,B 0,C 180,E1 33729.031,E2 33729.031} C_VEL
LIN {X 0,Y 729.535,Z 1146.971,A -85,B 0,C 180,E1 33727.831,E2 33727.831} C_VEL
LIN {X 0,Y 729.821,Z 1126.081,A -85,B 0,C 180,E1 33726.762,E2 33726.762} C_VEL
LIN {X 0,Y 730.164,Z 1104.69,A -85,B 0,C 180,E1 33725.831,E2 33725.831} C_VEL
LIN {X 0,Y 730.42,Z 1082.781,A -85,B 0,C 180,E1 33725.04,E2 33725.04} C_VEL
LIN {X 0,Y 730.699,Z 1058.742,A -85,B 0,C 180,E1 33724.345,E2 33724.345} C_VEL
LIN {X 0,Y 730.933,Z 1035.348,A -85,B 0,C 180,E1 33723.828,E2 33723.828} C_VEL
LIN {X 0,Y 731.074,Z 1012.289,A -85,B 0,C 180,E1 33723.471,E2 33723.471} C_VEL
LIN {X 0,Y 731.832,Z 741.585,A -85,B 0,C 180,E1 33720.541,E2 33720.541} C_VEL
LIN {X 0,Y 731.828,Z 675.245,A -85,B 0,C 180,E1 33719.806,E2 33719.806} C_VEL
LIN {X 0,Y 730.54,Z 669.44,A -85,B 0,C 180,E1 33719.667,E2 33719.667} C_VEL
LIN {X 0,Y 731.051,Z 628.375,A -85,B 0,C 180,E1 33716.831,E2 33716.831} C_VEL
LIN {X 0,Y 731.203,Z 618.258,A -85,B 0,C 180,E1 33716.113,E2 33716.113} C_VEL
LIN {X 0,Y 732.459,Z 618.876,A -85,B 0,C 180,E1 33715.967,E2 33715.967} C_VEL
LIN {X 0,Y 734.846,Z 617.58,A -85,B 0,C 180,E1 33715.692,E2 33715.692} C_VEL
LIN {X 0,Y 738.386,Z 613.102,A -85,B 0,C 180,E1 33715.292,E2 33715.292} C_VEL
LIN {X 0,Y 739.598,Z 611.305,A -85,B 0,C 180,E1 33715.157,E2 33715.157} C_VEL
LIN {X 0,Y 741.076,Z 613.18,A -85,B 0,C 180,E1 33714.993,E2 33714.993} C_VEL
LIN {X 0,Y 741.226,Z 772.926,A -85,B 0,C 180,E1 33714.976,E2 33714.976} C_VEL
LIN {X 0,Y 742.268,Z 783.454,A -85,B 0,C 180,E1 33714.862,E2 33714.862} C_VEL
LIN {X 0,Y 744.233,Z 792.46,A -85,B 0,C 180,E1 33714.647,E2 33714.647} C_VEL
LIN {X 0,Y 746.896,Z 800.081,A -85,B 0,C 180,E1 33714.339,E2 33714.339} C_VEL
LIN {X 0,Y 748.141,Z 804.754,A -85,B 0,C 180,E1 33714.006,E2 33714.006} C_VEL
LIN {X 0,Y 748.27,Z 808.2,A -85,B 0,C 180,E1 33713.61,E2 33713.61} C_VEL
LIN {X 0,Y 747.259,Z 810.451,A -85,B 0,C 180,E1 33713.147,E2 33713.147} C_VEL
LIN {X 0,Y 745.258,Z 811.1,A -85,B 0,C 180,E1 33712.67,E2 33712.67} C_VEL
LIN {X 0,Y 742.654,Z 810.109,A -85,B 0,C 180,E1 33712.216,E2 33712.216} C_VEL
LIN {X 0,Y 739.565,Z 807.368,A -85,B 0,C 180,E1 33711.768,E2 33711.768} C_VEL
LIN {X 0,Y 736.067,Z 802.065,A -85,B 0,C 180,E1 33711.229,E2 33711.229} C_VEL
LIN {X 0,Y 733.159,Z 794.074,A -85,B 0,C 180,E1 33710.527,E2 33710.527} C_VEL
LIN {X 0,Y 731.626,Z 783.393,A -85,B 0,C 180,E1 33709.694,E2 33709.694} C_VEL
LIN {X 0,Y 731.9,Z 730.722,A -85,B 0,C 180,E1 33705.896,E2 33705.896} C_VEL
LIN {X 0,Y 732.456,Z 693.929,A -85,B 0,C 180,E1 33703.151,E2 33703.151} C_VEL
LIN {X 0,Y 732.984,Z 658.752,A -85,B 0,C 180,E1 33700.434,E2 33700.434} C_VEL
LIN {X 0,Y 733.469,Z 623.876,A -85,B 0,C 180,E1 33697.642,E2 33697.642} C_VEL
LIN {X 0,Y 733.497,Z 610.269,A -85,B 0,C 180,E1 33696.515,E2 33696.515} C_VEL
LIN {X 0,Y 728.971,Z 599.925,A -85,B 0,C 180,E1 33695.273,E2 33695.273} C_VEL
LIN {X 0,Y 728.157,Z 597.27,A -85,B 0,C 180,E1 33694.955,E2 33694.955} C_VEL
LIN {X 0,Y 728.148,Z 597.281,A -85,B 0,C 180,E1 33691.917,E2 33691.917} C_VEL
LIN {X 0,Y 728.16,Z 597.281,A -85,B 0,C 180,E1 33688.905,E2 33688.905} C_VEL
LIN {X 0,Y 728.157,Z 597.282,A -85,B 0,C 180,E1 33685.921,E2 33685.921} C_VEL
LIN {X 0,Y 728.139,Z 597.282,A -85,B 0,C 180,E1 33683.04,E2 33683.04} C_VEL
LIN {X 0,Y 728.154,Z 597.277,A -85,B 0,C 180,E1 33680.078,E2 33680.078} C_VEL
LIN {X 0,Y 728.156,Z 597.275,A -85,B 0,C 180,E1 33677.089,E2 33677.089} C_VEL
LIN {X 0,Y 728.159,Z 597.275,A -85,B 0,C 180,E1 33673.986,E2 33673.986} C_VEL
LIN {X 0,Y 728.156,Z 597.274,A -85,B 0,C 180,E1 33670.924,E2 33670.924} C_VEL
LIN {X 0,Y 728.161,Z 597.275,A -85,B 0,C 180,E1 33667.813,E2 33667.813} C_VEL
LIN {X 0,Y 728.154,Z 597.276,A -85,B 0,C 180,E1 33664.726,E2 33664.726} C_VEL
LIN {X 0,Y 728.159,Z 597.276,A -85,B 0,C 180,E1 33661.652,E2 33661.652} C_VEL
LIN {X 0,Y 728.147,Z 597.28,A -85,B 0,C 180,E1 33658.662,E2 33658.662} C_VEL
LIN {X 0,Y 728.156,Z 597.282,A -85,B 0,C 180,E1 33655.747,E2 33655.747} C_VEL
LIN {X 0,Y 728.154,Z 597.279,A -85,B 0,C 180,E1 33652.822,E2 33652.822} C_VEL
LIN {X 0,Y 728.145,Z 597.277,A -85,B 0,C 180,E1 33649.876,E2 33649.876} C_VEL
LIN {X 0,Y 728.157,Z 597.275,A -85,B 0,C 180,E1 33646.904,E2 33646.904} C_VEL
LIN {X 0,Y 728.153,Z 597.28,A -85,B 0,C 180,E1 33646.369,E2 33646.369} C_VEL
LIN {X 0,Y 727.186,Z 597.406,A -85,B 0,C 180,E1 33645.763,E2 33645.763} C_VEL
LIN {X 0,Y 720.757,Z 598.198,A -85,B 0,C 180,E1 33644.066,E2 33644.066} C_VEL
LIN {X 0,Y 720.204,Z 598.266,A -85,B 0,C 180,E1 33643.624,E2 33643.624} C_VEL
LIN {X 0,Y 720.216,Z 598.264,A -85,B 0,C 180,E1 33640.621,E2 33640.621} C_VEL
LIN {X 0,Y 720.216,Z 598.265,A -85,B 0,C 180,E1 33637.555,E2 33637.555} C_VEL
LIN {X 0,Y 720.217,Z 598.265,A -85,B 0,C 180,E1 33634.472,E2 33634.472} C_VEL
LIN {X 0,Y 720.221,Z 598.265,A -85,B 0,C 180,E1 33631.382,E2 33631.382} C_VEL
LIN {X 0,Y 720.22,Z 598.265,A -85,B 0,C 180,E1 33628.253,E2 33628.253} C_VEL
LIN {X 0,Y 720.215,Z 598.266,A -85,B 0,C 180,E1 33625.208,E2 33625.208} C_VEL
LIN {X 0,Y 720.224,Z 598.266,A -85,B 0,C 180,E1 33622.147,E2 33622.147} C_VEL
LIN {X 0,Y 720.226,Z 598.27,A -85,B 0,C 180,E1 33619.164,E2 33619.164} C_VEL
LIN {X 0,Y 720.2,Z 598.265,A -85,B 0,C 180,E1 33616.213,E2 33616.213} C_VEL
LIN {X 0,Y 720.206,Z 598.267,A -85,B 0,C 180,E1 33613.299,E2 33613.299} C_VEL
LIN {X 0,Y 720.21,Z 598.265,A -85,B 0,C 180,E1 33610.415,E2 33610.415} C_VEL
LIN {X 0,Y 720.215,Z 598.263,A -85,B 0,C 180,E1 33607.349,E2 33607.349} C_VEL
LIN {X 0,Y 720.217,Z 598.263,A -85,B 0,C 180,E1 33604.304,E2 33604.304} C_VEL
LIN {X 0,Y 720.221,Z 598.268,A -85,B 0,C 180,E1 33601.186,E2 33601.186} C_VEL
LIN {X 0,Y 720.224,Z 598.346,A -85,B 0,C 180,E1 33599.252,E2 33599.252} C_VEL
LIN {X 0,Y 722.496,Z 607.147,A -85,B 0,C 180,E1 33598.608,E2 33598.608} C_VEL
LIN {X 0,Y 722.426,Z 644.907,A -85,B 0,C 180,E1 33596.199,E2 33596.199} C_VEL
LIN {X 0,Y 722.175,Z 683.033,A -85,B 0,C 180,E1 33593.758,E2 33593.758} C_VEL
LIN {X 0,Y 721.658,Z 729.036,A -85,B 0,C 180,E1 33590.813,E2 33590.813} C_VEL
LIN {X 0,Y 721.246,Z 774.992,A -85,B 0,C 180,E1 33587.923,E2 33587.923} C_VEL
LIN {X 0,Y 720.863,Z 823.042,A -85,B 0,C 180,E1 33584.95,E2 33584.95} C_VEL
LIN {X 0,Y 720.855,Z 831.116,A -85,B 0,C 180,E1 33584.478,E2 33584.478} C_VEL
LIN {X 0,Y 721.266,Z 838.997,A -85,B 0,C 180,E1 33584.39,E2 33584.39} C_VEL
LIN {X 0,Y 720.968,Z 1001.06,A -85,B 0,C 180,E1 33582.74,E2 33582.74} C_VEL
LIN {X 0,Y 720.881,Z 1018.915,A -85,B 0,C 180,E1 33582.401,E2 33582.401} C_VEL
LIN {X 0,Y 720.754,Z 1035.787,A -85,B 0,C 180,E1 33581.928,E2 33581.928} C_VEL
LIN {X 0,Y 720.619,Z 1051.895,A -85,B 0,C 180,E1 33581.322,E2 33581.322} C_VEL
LIN {X 0,Y 720.481,Z 1067.028,A -85,B 0,C 180,E1 33580.595,E2 33580.595} C_VEL
LIN {X 0,Y 720.328,Z 1081.751,A -85,B 0,C 180,E1 33579.708,E2 33579.708} C_VEL
LIN {X 0,Y 720.201,Z 1095.411,A -85,B 0,C 180,E1 33578.694,E2 33578.694} C_VEL
LIN {X 0,Y 720.1,Z 1106.783,A -85,B 0,C 180,E1 33577.659,E2 33577.659} C_VEL
LIN {X 0,Y 720.019,Z 1117.475,A -85,B 0,C 180,E1 33576.457,E2 33576.457} C_VEL
LIN {X 0,Y 719.965,Z 1126.545,A -85,B 0,C 180,E1 33575.178,E2 33575.178} C_VEL
LIN {X 0,Y 719.937,Z 1133.578,A -85,B 0,C 180,E1 33573.901,E2 33573.901} C_VEL
LIN {X 0,Y 719.921,Z 1139.052,A -85,B 0,C 180,E1 33572.546,E2 33572.546} C_VEL
LIN {X 0,Y 719.914,Z 1142.685,A -85,B 0,C 180,E1 33571.193,E2 33571.193} C_VEL
LIN {X 0,Y 719.915,Z 1144.675,A -85,B 0,C 180,E1 33569.76,E2 33569.76} C_VEL
LIN {X 0,Y 719.915,Z 1144.853,A -85,B 0,C 180,E1 33568.407,E2 33568.407} C_VEL
LIN {X 0,Y 719.917,Z 1143.226,A -85,B 0,C 180,E1 33566.992,E2 33566.992} C_VEL
LIN {X 0,Y 719.92,Z 1139.855,A -85,B 0,C 180,E1 33565.618,E2 33565.618} C_VEL
LIN {X 0,Y 719.93,Z 1134.713,A -85,B 0,C 180,E1 33564.26,E2 33564.26} C_VEL
LIN {X 0,Y 719.958,Z 1128.063,A -85,B 0,C 180,E1 33562.979,E2 33562.979} C_VEL
LIN {X 0,Y 720.006,Z 1120.005,A -85,B 0,C 180,E1 33561.775,E2 33561.775} C_VEL
LIN {X 0,Y 720.074,Z 1109.828,A -85,B 0,C 180,E1 33560.568,E2 33560.568} C_VEL
LIN {X 0,Y 720.177,Z 1097.786,A -85,B 0,C 180,E1 33559.417,E2 33559.417} C_VEL
LIN {X 0,Y 720.301,Z 1085.083,A -85,B 0,C 180,E1 33558.428,E2 33558.428} C_VEL
LIN {X 0,Y 720.436,Z 1070.973,A -85,B 0,C 180,E1 33557.536,E2 33557.536} C_VEL
LIN {X 0,Y 720.571,Z 1055.846,A -85,B 0,C 180,E1 33556.763,E2 33556.763} C_VEL
LIN {X 0,Y 720.719,Z 1039.642,A -85,B 0,C 180,E1 33556.112,E2 33556.112} C_VEL
LIN {X 0,Y 720.857,Z 1022.633,A -85,B 0,C 180,E1 33555.6,E2 33555.6} C_VEL
LIN {X 0,Y 720.958,Z 1004.749,A -85,B 0,C 180,E1 33555.227,E2 33555.227} C_VEL
LIN {X 0,Y 721.018,Z 981.855,A -85,B 0,C 180,E1 33554.956,E2 33554.956} C_VEL
LIN {X 0,Y 721.04,Z 832.597,A -85,B 0,C 180,E1 33553.451,E2 33553.451} C_VEL
LIN {X 0,Y 720.804,Z 830.126,A -85,B 0,C 180,E1 33553.395,E2 33553.395} C_VEL
LIN {X 0,Y 721.178,Z 782.897,A -85,B 0,C 180,E1 33550.479,E2 33550.479} C_VEL
LIN {X 0,Y 721.625,Z 734.269,A -85,B 0,C 180,E1 33547.429,E2 33547.429} C_VEL
LIN {X 0,Y 722.086,Z 688.973,A -85,B 0,C 180,E1 33544.535,E2 33544.535} C_VEL
LIN {X 0,Y 722.446,Z 649.685,A -85,B 0,C 180,E1 33542.009,E2 33542.009} C_VEL
LIN {X 0,Y 722.531,Z 606.503,A -85,B 0,C 180,E1 33539.248,E2 33539.248} C_VEL
LIN {X 0,Y 720.209,Z 598.271,A -85,B 0,C 180,E1 33538.631,E2 33538.631} C_VEL
LIN {X 0,Y 720.216,Z 598.26,A -85,B 0,C 180,E1 33535.69,E2 33535.69} C_VEL
LIN {X 0,Y 720.219,Z 598.264,A -85,B 0,C 180,E1 33532.572,E2 33532.572} C_VEL
LIN {X 0,Y 720.204,Z 598.261,A -85,B 0,C 180,E1 33529.659,E2 33529.659} C_VEL
LIN {X 0,Y 720.202,Z 598.267,A -85,B 0,C 180,E1 33526.793,E2 33526.793} C_VEL
LIN {X 0,Y 720.203,Z 598.264,A -85,B 0,C 180,E1 33523.899,E2 33523.899} C_VEL
LIN {X 0,Y 720.212,Z 598.266,A -85,B 0,C 180,E1 33520.942,E2 33520.942} C_VEL
LIN {X 0,Y 720.223,Z 598.263,A -85,B 0,C 180,E1 33517.948,E2 33517.948} C_VEL
LIN {X 0,Y 720.217,Z 598.265,A -85,B 0,C 180,E1 33514.865,E2 33514.865} C_VEL
LIN {X 0,Y 720.208,Z 598.269,A -85,B 0,C 180,E1 33511.935,E2 33511.935} C_VEL
LIN {X 0,Y 720.199,Z 598.27,A -85,B 0,C 180,E1 33508.994,E2 33508.994} C_VEL
LIN {X 0,Y 720.205,Z 598.322,A -85,B 0,C 180,E1 33507.964,E2 33507.964} C_VEL
LIN {X 0,Y 721.084,Z 601.352,A -85,B 0,C 180,E1 33507.691,E2 33507.691} C_VEL
LIN {X 0,Y 725.059,Z 609.906,A -85,B 0,C 180,E1 33507.408,E2 33507.408} C_VEL
LIN {X 0,Y 724.188,Z 866.771,A -85,B 0,C 180,E1 33504.593,E2 33504.593} C_VEL
LIN {X 0,Y 723.888,Z 946.875,A -85,B 0,C 180,E1 33503.706,E2 33503.706} C_VEL
LIN {X 0,Y 723.654,Z 971.092,A -85,B 0,C 180,E1 33503.293,E2 33503.293} C_VEL
LIN {X 0,Y 723.392,Z 993.211,A -85,B 0,C 180,E1 33502.77,E2 33502.77} C_VEL
LIN {X 0,Y 723.048,Z 1014.162,A -85,B 0,C 180,E1 33502.138,E2 33502.138} C_VEL
LIN {X 0,Y 722.744,Z 1035.953,A -85,B 0,C 180,E1 33501.337,E2 33501.337} C_VEL
LIN {X 0,Y 722.312,Z 1057.622,A -85,B 0,C 180,E1 33500.374,E2 33500.374} C_VEL
LIN {X 0,Y 721.936,Z 1078.35,A -85,B 0,C 180,E1 33499.289,E2 33499.289} C_VEL
LIN {X 0,Y 721.545,Z 1098.703,A -85,B 0,C 180,E1 33498.042,E2 33498.042} C_VEL
LIN {X 0,Y 721.155,Z 1117.777,A -85,B 0,C 180,E1 33496.679,E2 33496.679} C_VEL
LIN {X 0,Y 720.844,Z 1135.708,A -85,B 0,C 180,E1 33495.199,E2 33495.199} C_VEL
LIN {X 0,Y 720.583,Z 1152.03,A -85,B 0,C 180,E1 33493.644,E2 33493.644} C_VEL
LIN {X 0,Y 720.354,Z 1166.723,A -85,B 0,C 180,E1 33492.017,E2 33492.017} C_VEL
LIN {X 0,Y 720.179,Z 1179.879,A -85,B 0,C 180,E1 33490.318,E2 33490.318} C_VEL
LIN {X 0,Y 720.07,Z 1191.596,A -85,B 0,C 180,E1 33488.545,E2 33488.545} C_VEL
LIN {X 0,Y 719.998,Z 1201.214,A -85,B 0,C 180,E1 33486.779,E2 33486.779} C_VEL
LIN {X 0,Y 719.952,Z 1209.446,A -85,B 0,C 180,E1 33484.94,E2 33484.94} C_VEL
LIN {X 0,Y 719.925,Z 1215.557,A -85,B 0,C 180,E1 33483.185,E2 33483.185} C_VEL
LIN {X 0,Y 719.909,Z 1220.615,A -85,B 0,C 180,E1 33481.194,E2 33481.194} C_VEL
